  MoveL 1318 to (27.18, 67.36, -94.62) mm, rotated rx -11.83 ry -17.7 rz 126.62 deg; joints [8.101, -41.729, 125.318, 236.035, 70.646, -43.276, 143.741]
  MoveL 1319 to (26.72, 68.02, -94.62) mm, rotated rx -11.83 ry -17.7 rz 126.62 deg; joints [8.127, -41.741, 125.362, 236.053, 70.666, -43.25, 143.741]
  MoveL 1320 to (26.37, 68.63, -94.62) mm, rotated rx -11.83 ry -17.7 rz 126.62 deg; joints [8.149, -41.755, 125.404, 236.067, 70.684, -43.226, 143.741]
  MoveL 1321 to (26.15, 69.22, -94.62) mm, rotated rx -11.83 ry -17.7 rz 126.62 deg; joints [8.165, -41.771, 125.447, 236.075, 70.7, -43.204, 143.741]
  MoveL 1322 to (25.94, 69.86, -94.6) mm, rotated rx -11.83 ry -17.7 rz 126.62 deg; joints [8.181, -41.791, 125.494, 236.083, 70.717, -43.181, 143.741]
  MoveL 1323 to (25.74, 70.59, -94.56) mm, rotated rx -11.83 ry -17.7 rz 126.62 deg; joints [8.198, -41.815, 125.548, 236.092, 70.735, -43.156, 143.741]
  MoveL 1324 to (25.25, 72.63, -94.56) mm, rotated rx -11.83 ry -17.7 rz 126.62 deg; joints [8.24, -41.878, 125.7, 236.109, 70.789, -43.08, 143.741]
  MoveL 1325 to (25.13, 73.06, -94.54) mm, rotated rx -11.83 ry -17.7 rz 126.62 deg; joints [8.25, -41.892, 125.732, 236.114, 70.799, -43.066, 143.741]
  MoveL 1326 to (24.89, 74.08, -94.54) mm, rotated rx -11.83 ry -17.7 rz 126.62 deg; joints [8.271, -41.924, 125.808, 236.122, 70.826, -43.028, 143.741]
  MoveL 1327 to (24.77, 74.57, -94.54) mm, rotated rx -11.83 ry -17.7 rz 126.62 deg; joints [8.281, -41.939, 125.844, 236.127, 70.839, -43.01, 143.741]
  MoveL 1328 to (24.64, 75.04, -94.52) mm, rotated rx -11.83 ry -17.7 rz 126.62 deg; joints [8.292, -41.954, 125.879, 236.132, 70.85, -42.993, 143.741]
  MoveL 1329 to (24.51, 75.5, -94.49) mm, rotated rx -11.83 ry -17.7 rz 126.62 deg; joints [8.303, -41.97, 125.913, 236.138, 70.862, -42.978, 143.741]
  MoveL 1330 to (24.37, 75.91, -94.43) mm, rotated rx -11.83 ry -17.7 rz 126.62 deg; joints [8.314, -41.985, 125.942, 236.145, 70.871, -42.966, 143.741]
  MoveL 1331 to (24.24, 76.37, -94.39) mm, rotated rx -11.83 ry -17.7 rz 126.62 deg; joints [8.325, -42, 125.975, 236.151, 70.882, -42.951, 143.741]
  MoveL 1332 to (24.11, 76.85, -94.37) mm, rotated rx -11.83 ry -17.7 rz 126.62 deg; joints [8.336, -42.016, 126.011, 236.156, 70.893, -42.935, 143.741]
  MoveL 1333 to (23.99, 77.34, -94.37) mm, rotated rx -11.83 ry -17.7 rz 126.62 deg; joints [8.347, -42.031, 126.047, 236.161, 70.906, -42.917, 143.741]
  MoveL 1334 to (23.86, 77.81, -94.35) mm, rotated rx -11.83 ry -17.7 rz 126.62 deg; joints [8.357, -42.047, 126.082, 236.167, 70.918, -42.9, 143.741]
  MoveL 1335 to (23.72, 78.27, -94.31) mm, rotated rx -11.83 ry -17.7 rz 126.62 deg; joints [8.369, -42.062, 126.116, 236.173, 70.929, -42.885, 143.741]
  MoveL 1336 to (23.58, 78.68, -94.26) mm, rotated rx -11.83 ry -17.7 rz 126.62 deg; joints [8.38, -42.077, 126.145, 236.18, 70.938, -42.873, 143.741]
  MoveL 1337 to (23.43, 79.11, -94.2) mm, rotated rx -11.83 ry -17.7 rz 126.62 deg; joints [8.392, -42.092, 126.176, 236.188, 70.948, -42.86, 143.741]
  MoveL 1338 to (23.03, 80.5, -94.12) mm, rotated rx -11.83 ry -17.7 rz 126.62 deg; joints [8.425, -42.138, 126.277, 236.205, 70.982, -42.813, 143.741]
  MoveL 1339 to (22.85, 81.66, -94.25) mm, rotated rx -11.83 ry -17.7 rz 126.62 deg; joints [8.443, -42.168, 126.366, 236.208, 71.015, -42.763, 143.741]
  MoveL 1340 to (22.88, 82.6, -94.58) mm, rotated rx -11.83 ry -17.7 rz 126.62 deg; joints [8.447, -42.184, 126.441, 236.194, 71.049, -42.711, 143.741]
  MoveL 1341 to (22.98, 82.99, -94.83) mm, rotated rx -11.83 ry -17.7 rz 126.62 deg; joints [8.444, -42.187, 126.475, 236.182, 71.066, -42.683, 143.741]
  MoveL 1342 to (23.13, 83.33, -95.13) mm, rotated rx -11.83 ry -17.7 rz 126.62 deg; joints [8.436, -42.185, 126.505, 236.165, 71.083, -42.655, 143.741]
  MoveL 1343 to (23.59, 83.83, -95.89) mm, rotated rx -11.83 ry -17.7 rz 126.62 deg; joints [8.41, -42.172, 126.556, 236.121, 71.116, -42.597, 143.741]
  MoveL 1344 to (24.27, 84.12, -96.86) mm, rotated rx -11.83 ry -17.7 rz 126.62 deg; joints [8.37, -42.143, 126.594, 236.061, 71.15, -42.536, 143.741]
  MoveL 1345 to (26.28, 84.03, -99.42) mm, rotated rx -11.83 ry -17.7 rz 126.62 deg; joints [8.244, -42.041, 126.632, 235.894, 71.219, -42.407, 143.741]
  MoveL 1346 to (28.47, 83.17, -102.03) mm, rotated rx -11.83 ry -17.7 rz 126.62 deg; joints [8.102, -41.913, 126.613, 235.72, 71.269, -42.304, 143.741]
  MoveL 1347 to (29.36, 82.49, -103.06) mm, rotated rx -11.83 ry -17.7 rz 126.62 deg; joints [8.041, -41.851, 126.579, 235.65, 71.28, -42.276, 143.741]
  MoveL 1348 to (30.13, 81.66, -103.9) mm, rotated rx -11.83 ry -17.7 rz 126.62 deg; joints [7.987, -41.791, 126.529, 235.592, 71.282, -42.264, 143.741]
  MoveL 1349 to (30.76, 80.65, -104.55) mm, rotated rx -11.83 ry -17.7 rz 126.62 deg; joints [7.94, -41.732, 126.464, 235.546, 71.275, -42.267, 143.741]
  MoveL 1350 to (31.27, 79.49, -105.02) mm, rotated rx -11.83 ry -17.7 rz 126.62 deg; joints [7.899, -41.675, 126.383, 235.511, 71.258, -42.286, 143.741]
  MoveL 1351 to (31.64, 78.15, -105.3) mm, rotated rx -11.83 ry -17.7 rz 126.62 deg; joints [7.865, -41.62, 126.286, 235.489, 71.232, -42.32, 143.741]
  MoveL 1352 to (31.88, 76.66, -105.39) mm, rotated rx -11.83 ry -17.7 rz 126.62 deg; joints [7.838, -41.566, 126.173, 235.478, 71.196, -42.37, 143.741]
  MoveL 1353 to (32.24, 73.52, -105.39) mm, rotated rx -11.83 ry -17.7 rz 126.62 deg; joints [7.791, -41.46, 125.932, 235.468, 71.116, -42.484, 143.741]
  MoveL 1354 to (32.31, 72.97, -105.41) mm, rotated rx -11.83 ry -17.7 rz 126.62 deg; joints [7.782, -41.441, 125.89, 235.466, 71.103, -42.504, 143.741]
  MoveL 1355 to (32.41, 72.36, -105.44) mm, rotated rx -11.83 ry -17.7 rz 126.62 deg; joints [7.772, -41.418, 125.844, 235.462, 71.088, -42.524, 143.741]
  MoveL 1356 to (32.55, 71.61, -105.54) mm, rotated rx -11.83 ry -17.7 rz 126.62 deg; joints [7.757, -41.389, 125.788, 235.454, 71.072, -42.547, 143.741]
  MoveL 1357 to (32.65, 71, -105.58) mm, rotated rx -11.83 ry -17.7 rz 126.62 deg; joints [7.746, -41.367, 125.741, 235.45, 71.057, -42.567, 143.741]
  MoveL 1358 to (32.72, 70.46, -105.59) mm, rotated rx -11.83 ry -17.7 rz 126.62 deg; joints [7.737, -41.348, 125.7, 235.447, 71.044, -42.586, 143.741]
  MoveL 1359 to (32.78, 69.96, -105.6) mm, rotated rx -11.83 ry -17.7 rz 126.62 deg; joints [7.729, -41.331, 125.662, 235.445, 71.031, -42.604, 143.741]
  MoveL 1360 to (32.85, 69.5, -105.61) mm, rotated rx -11.83 ry -17.7 rz 126.62 deg; joints [7.722, -41.315, 125.627, 235.443, 71.02, -42.62, 143.741]
  MoveL 1361 to (33.08, 67.46, -105.62) mm, rotated rx -11.83 ry -17.7 rz 126.62 deg; joints [7.691, -41.245, 125.47, 235.437, 70.968, -42.694, 143.741]
  MoveL 1362 to (33.16, 66.95, -105.66) mm, rotated rx -11.83 ry -17.7 rz 126.62 deg; joints [7.682, -41.227, 125.432, 235.433, 70.956, -42.711, 143.741]
  MoveL 1363 to (33.26, 66.49, -105.71) mm, rotated rx -11.83 ry -17.7 rz 126.62 deg; joints [7.673, -41.209, 125.397, 235.429, 70.945, -42.725, 143.741]
  MoveL 1364 to (33.36, 66.04, -105.78) mm, rotated rx -11.83 ry -17.7 rz 126.62 deg; joints [7.663, -41.191, 125.363, 235.423, 70.936, -42.738, 143.741]
  MoveL 1365 to (33.49, 65.57, -105.84) mm, rotated rx -11.83 ry -17.7 rz 126.62 deg; joints [7.652, -41.174, 125.329, 235.416, 70.925, -42.753, 143.741]
  MoveL 1366 to (33.66, 65.05, -105.88) mm, rotated rx -11.83 ry -17.7 rz 126.62 deg; joints [7.639, -41.157, 125.29, 235.41, 70.912, -42.771, 143.741]
  MoveL 1367 to (33.95, 64.44, -105.88) mm, rotated rx -11.83 ry -17.7 rz 126.62 deg; joints [7.62, -41.142, 125.247, 235.399, 70.894, -42.794, 143.741]
  MoveL 1368 to (34.35, 63.78, -105.88) mm, rotated rx -11.83 ry -17.7 rz 126.62 deg; joints [7.596, -41.128, 125.201, 235.383, 70.874, -42.82, 143.741]
  MoveL 1369 to (34.26, 65.71, -107.44) mm, rotated rx -11.83 ry -17.7 rz 126.62 deg; joints [7.597, -41.106, 125.358, 235.333, 70.976, -42.664, 143.741]
  MoveL 1370 to (35.81, 63.93, -107.57) mm, rotated rx -11.83 ry -17.7 rz 126.62 deg; joints [7.51, -41.073, 125.243, 235.268, 70.922, -42.731, 143.741]
  MoveL 1371 to (37.27, 62.24, -107.68) mm, rotated rx -11.83 ry -17.7 rz 126.62 deg; joints [7.428, -41.043, 125.134, 235.208, 70.869, -42.795, 143.741]
  MoveL 1372 to (38.69, 60.61, -107.84) mm, rotated rx -11.83 ry -17.7 rz 126.62 deg; joints [7.348, -41.012, 125.029, 235.148, 70.821, -42.854, 143.741]
  MoveL 1373 to (40.09, 59, -107.95) mm, rotated rx -11.83 ry -17.7 rz 126.62 deg; joints [7.27, -40.982, 124.924, 235.09, 70.771, -42.915, 143.741]
  MoveL 1374 to (41.49, 57.38, -108.06) mm, rotated rx -11.83 ry -17.7 rz 126.62 deg; joints [7.193, -40.953, 124.818, 235.033, 70.72, -42.976, 143.741]
  MoveL 1375 to (42.89, 55.78, -108.28) mm, rotated rx -11.83 ry -17.7 rz 126.62 deg; joints [7.113, -40.918, 124.713, 234.972, 70.674, -43.031, 143.741]
  MoveL 1376 to (44.29, 54.16, -108.5) mm, rotated rx -11.83 ry -17.7 rz 126.62 deg; joints [7.034, -40.881, 124.608, 234.912, 70.627, -43.085, 143.741]
  MoveL 1377 to (45.68, 52.54, -108.62) mm, rotated rx -11.83 ry -17.7 rz 126.62 deg; joints [6.957, -40.851, 124.501, 234.856, 70.576, -43.146, 143.741]
  MoveL 1378 to (47.06, 50.91, -108.62) mm, rotated rx -11.83 ry -17.7 rz 126.62 deg; joints [6.882, -40.827, 124.393, 234.804, 70.521, -43.214, 143.741]
  MoveL 1379 to (48.44, 49.29, -108.73) mm, rotated rx -11.83 ry -17.7 rz 126.62 deg; joints [6.806, -40.796, 124.286, 234.748, 70.47, -43.275, 143.741]
  MoveL 1380 to (49.85, 47.65, -108.93) mm, rotated rx -11.83 ry -17.7 rz 126.62 deg; joints [6.727, -40.759, 124.177, 234.689, 70.421, -43.332, 143.741]
  MoveL 1381 to (51.15, 46.11, -109.11) mm, rotated rx -11.83 ry -17.7 rz 126.62 deg; joints [6.654, -40.725, 124.075, 234.635, 70.374, -43.386, 143.741]
  MoveL 1382 to (52.35, 44.7, -109.33) mm, rotated rx -11.83 ry -17.7 rz 126.62 deg; joints [6.587, -40.691, 123.981, 234.583, 70.334, -43.433, 143.741]
  MoveL 1383 to (53.63, 43.2, -109.42) mm, rotated rx -11.83 ry -17.7 rz 126.62 deg; joints [6.517, -40.663, 123.881, 234.533, 70.285, -43.49, 143.741]
  MoveL 1384 to (54.98, 41.6, -109.43) mm, rotated rx -11.83 ry -17.7 rz 126.62 deg; joints [6.444, -40.637, 123.774, 234.483, 70.231, -43.555, 143.741]
  MoveL 1385 to (56.72, 39.52, -109.53) mm, rotated rx -11.83 ry -17.7 rz 126.62 deg; joints [6.35, -40.599, 123.634, 234.417, 70.163, -43.636, 143.741]
  MoveL 1386 to (58.02, 37.96, -109.74) mm, rotated rx -11.83 ry -17.7 rz 126.62 deg; joints [6.277, -40.561, 123.529, 234.363, 70.116, -43.689, 143.741]
  MoveL 1387 to (59.42, 36.26, -109.94) mm, rotated rx -11.83 ry -17.7 rz 126.62 deg; joints [6.199, -40.521, 123.413, 234.306, 70.064, -43.748, 143.741]
  MoveL 1388 to (60.7, 34.69, -110.23) mm, rotated rx -11.83 ry -17.7 rz 126.62 deg; joints [6.127, -40.479, 123.307, 234.251, 70.02, -43.797, 143.741]
  MoveL 1389 to (61.97, 33.17, -110.36) mm, rotated rx -11.83 ry -17.7 rz 126.62 deg; joints [6.058, -40.446, 123.204, 234.201, 69.971, -43.853, 143.741]
  MoveL 1390 to (63.32, 31.57, -110.38) mm, rotated rx -11.83 ry -17.7 rz 126.62 deg; joints [5.986, -40.42, 123.095, 234.152, 69.916, -43.918, 143.741]
  MoveL 1391 to (64.43, 30.19, -110.6) mm, rotated rx -11.83 ry -17.7 rz 126.62 deg; joints [5.924, -40.382, 123, 234.106, 69.876, -43.963, 143.741]
  Set speed (1000.0 mm/s)
  MoveL 1392 to (88.04, 19.17, -110.6) mm, rotated rx -11.83 ry -17.7 rz 126.62 deg; joints [4.825, -40.56, 122.428, 233.209, 69.312, -44.514, 143.741]
  Set speed (1000.0 mm/s)
  MoveL 1393 to (85.28, 13.25, -121.79) mm, rotated rx -11.83 ry -17.7 rz 126.62 deg; joints [4.742, -39.632, 121.949, 232.99, 69.573, -44.122, 143.741]
  Set speed (100.0 mm/s)
  MoveL 1394 to (67, 21.77, -121.79) mm, rotated rx -11.83 ry -17.7 rz 126.62 deg; joints [5.589, -39.492, 122.393, 233.681, 70.009, -43.693, 143.741]
  MoveL 1395 to (65.84, 23.56, -121.79) mm, rotated rx -11.83 ry -17.7 rz 126.62 deg; joints [5.653, -39.53, 122.521, 233.72, 70.068, -43.62, 143.741]
  MoveL 1396 to (64.64, 25.44, -121.69) mm, rotated rx -11.83 ry -17.7 rz 126.62 deg; joints [5.721, -39.575, 122.656, 233.764, 70.128, -43.55, 143.741]
  MoveL 1397 to (63.4, 27.44, -121.4) mm, rotated rx -11.83 ry -17.7 rz 126.62 deg; joints [5.795, -39.635, 122.798, 233.814, 70.183, -43.484, 143.741]
  MoveL 1398 to (62.23, 29.36, -121.05) mm, rotated rx -11.83 ry -17.7 rz 126.62 deg; joints [5.866, -39.697, 122.935, 233.865, 70.234, -43.425, 143.741]
  MoveL 1399 to (61.12, 31.11, -120.86) mm, rotated rx -11.83 ry -17.7 rz 126.62 deg; joints [5.93, -39.745, 123.059, 233.909, 70.286, -43.364, 143.741]
  MoveL 1400 to (60.07, 32.75, -120.73) mm, rotated rx -11.83 ry -17.7 rz 126.62 deg; joints [5.991, -39.787, 123.175, 233.949, 70.335, -43.305, 143.741]
  MoveL 1401 to (58.95, 34.47, -120.68) mm, rotated rx -11.83 ry -17.7 rz 126.62 deg; joints [6.055, -39.825, 123.297, 233.99, 70.39, -43.238, 143.741]
  MoveL 1402 to (57.78, 36.26, -120.66) mm, rotated rx -11.83 ry -17.7 rz 126.62 deg; joints [6.12, -39.862, 123.423, 234.031, 70.448, -43.167, 143.741]
  MoveL 1403 to (56.63, 38.04, -120.54) mm, rotated rx -11.83 ry -17.7 rz 126.62 deg; joints [6.187, -39.905, 123.548, 234.075, 70.502, -43.101, 143.741]
  MoveL 1404 to (55.38, 39.96, -120.28) mm, rotated rx -11.83 ry -17.7 rz 126.62 deg; joints [6.261, -39.959, 123.682, 234.127, 70.556, -43.036, 143.741]
  MoveL 1405 to (54.07, 41.97, -120.09) mm, rotated rx -11.83 ry -17.7 rz 126.62 deg; joints [6.338, -40.01, 123.823, 234.18, 70.615, -42.965, 143.741]
  MoveL 1406 to (52.79, 43.92, -119.89) mm, rotated rx -11.83 ry -17.7 rz 126.62 deg; joints [6.413, -40.061, 123.959, 234.232, 70.672, -42.896, 143.741]
  MoveL 1407 to (51.62, 45.7, -119.78) mm, rotated rx -11.83 ry -17.7 rz 126.62 deg; joints [6.481, -40.103, 124.083, 234.278, 70.726, -42.83, 143.741]
  MoveL 1408 to (49.29, 49.23, -119.51) mm, rotated rx -11.83 ry -17.7 rz 126.62 deg; joints [6.618, -40.187, 124.328, 234.371, 70.83, -42.701, 143.741]
  MoveL 1409 to (48.1, 51.05, -119.44) mm, rotated rx -11.83 ry -17.7 rz 126.62 deg; joints [6.687, -40.227, 124.454, 234.417, 70.887, -42.631, 143.741]
  MoveL 1410 to (46.91, 52.82, -119.22) mm, rotated rx -11.83 ry -17.7 rz 126.62 deg; joints [6.758, -40.273, 124.575, 234.468, 70.936, -42.571, 143.741]
  MoveL 1411 to (45.73, 54.57, -119.06) mm, rotated rx -11.83 ry -17.7 rz 126.62 deg; joints [6.828, -40.316, 124.696, 234.517, 70.987, -42.508, 143.741]
  MoveL 1412 to (44.55, 56.32, -118.87) mm, rotated rx -11.83 ry -17.7 rz 126.62 deg; joints [6.898, -40.359, 124.816, 234.567, 71.036, -42.446, 143.741]
  MoveL 1413 to (43.34, 58.13, -118.78) mm, rotated rx -11.83 ry -17.7 rz 126.62 deg; joints [6.969, -40.399, 124.94, 234.615, 71.091, -42.377, 143.741]
  MoveL 1414 to (42.07, 60.01, -118.65) mm, rotated rx -11.83 ry -17.7 rz 126.62 deg; joints [7.044, -40.441, 125.068, 234.667, 71.147, -42.308, 143.741]
  MoveL 1415 to (41.03, 61.61, -118.59) mm, rotated rx -11.83 ry -17.7 rz 126.62 deg; joints [7.105, -40.476, 125.178, 234.708, 71.195, -42.246, 143.741]
  MoveL 1416 to (40.47, 61.24, -117.71) mm, rotated rx -11.83 ry -17.7 rz 126.62 deg; joints [7.138, -40.5, 125.138, 234.76, 71.16, -42.303, 143.741]
  MoveL 1417 to (40.45, 60.88, -117.3) mm, rotated rx -11.83 ry -17.7 rz 126.62 deg; joints [7.142, -40.511, 125.108, 234.775, 71.137, -42.339, 143.741]
  MoveL 1418 to (40.41, 60.83, -117.02) mm, rotated rx -11.83 ry -17.7 rz 126.62 deg; joints [7.147, -40.524, 125.102, 234.785, 71.126, -42.356, 143.741]
  MoveL 1419 to (40.36, 61.15, -116.9) mm, rotated rx -11.83 ry -17.7 rz 126.62 deg; joints [7.154, -40.542, 125.127, 234.79, 71.131, -42.35, 143.741]
  MoveL 1420 to (40.33, 61.6, -116.84) mm, rotated rx -11.83 ry -17.7 rz 126.62 deg; joints [7.16, -40.561, 125.162, 234.792, 71.141, -42.337, 143.741]
  MoveL 1421 to (40.31, 62.16, -116.81) mm, rotated rx -11.83 ry -17.7 rz 126.62 deg; joints [7.167, -40.583, 125.206, 234.793, 71.154, -42.318, 143.741]
  MoveL 1422 to (40.3, 62.86, -116.77) mm, rotated rx -11.83 ry -17.7 rz 126.62 deg; joints [7.175, -40.61, 125.26, 234.793, 71.17, -42.295, 143.741]
  MoveL 1423 to (40.29, 63.49, -116.74) mm, rotated rx -11.83 ry -17.7 rz 126.62 deg; joints [7.181, -40.634, 125.31, 234.793, 71.185, -42.273, 143.741]
  MoveL 1424 to (40.3, 64.02, -116.74) mm, rotated rx -11.83 ry -17.7 rz 126.62 deg; joints [7.186, -40.654, 125.352, 234.791, 71.199, -42.254, 143.741]
  MoveL 1425 to (40.29, 64.5, -116.73) mm, rotated rx -11.83 ry -17.7 rz 126.62 deg; joints [7.191, -40.672, 125.39, 234.791, 71.21, -42.237, 143.741]
  MoveL 1426 to (40.25, 65.54, -116.65) mm, rotated rx -11.83 ry -17.7 rz 126.62 deg; joints [7.204, -40.714, 125.471, 234.793, 71.234, -42.204, 143.741]
  MoveL 1427 to (40.22, 66.1, -116.6) mm, rotated rx -11.83 ry -17.7 rz 126.62 deg; joints [7.211, -40.736, 125.515, 234.794, 71.247, -42.186, 143.741]
  MoveL 1428 to (40.18, 66.61, -116.53) mm, rotated rx -11.83 ry -17.7 rz 126.62 deg; joints [7.218, -40.758, 125.554, 234.797, 71.258, -42.171, 143.741]
  MoveL 1429 to (40.14, 67.07, -116.46) mm, rotated rx -11.83 ry -17.7 rz 126.62 deg; joints [7.226, -40.778, 125.59, 234.8, 71.267, -42.158, 143.741]
  MoveL 1430 to (40.1, 67.54, -116.4) mm, rotated rx -11.83 ry -17.7 rz 126.62 deg; joints [7.232, -40.797, 125.625, 234.802, 71.277, -42.144, 143.741]
  MoveL 1431 to (40.09, 68.02, -116.37) mm, rotated rx -11.83 ry -17.7 rz 126.62 deg; joints [7.238, -40.816, 125.663, 234.803, 71.288, -42.129, 143.741]
  MoveL 1432 to (40.08, 68.54, -116.35) mm, rotated rx -11.83 ry -17.7 rz 126.62 deg; joints [7.244, -40.836, 125.704, 234.803, 71.301, -42.111, 143.741]
  MoveL 1433 to (40.12, 72.21, -116.35) mm, rotated rx -11.83 ry -17.7 rz 126.62 deg; joints [7.277, -40.971, 125.994, 234.793, 71.393, -41.979, 143.741]
  MoveL 1434 to (40.25, 73.83, -116.37) mm, rotated rx -11.83 ry -17.7 rz 126.62 deg; joints [7.286, -41.031, 126.123, 234.784, 71.433, -41.92, 143.741]
  MoveL 1435 to (40.39, 74.39, -116.4) mm, rotated rx -11.83 ry -17.7 rz 126.62 deg; joints [7.285, -41.054, 126.169, 234.776, 71.447, -41.899, 143.741]
  MoveL 1436 to (40.57, 74.79, -116.43) mm, rotated rx -11.83 ry -17.7 rz 126.62 deg; joints [7.281, -41.071, 126.204, 234.767, 71.456, -41.884, 143.741]
  MoveL 1437 to (40.78, 75.06, -116.47) mm, rotated rx -11.83 ry -17.7 rz 126.62 deg; joints [7.273, -41.084, 126.229, 234.756, 71.462, -41.874, 143.741]
  MoveL 1438 to (40.9, 75.14, -116.5) mm, rotated rx -11.83 ry -17.7 rz 126.62 deg; joints [7.268, -41.089, 126.237, 234.75, 71.464, -41.87, 143.741]
  MoveL 1439 to (41.03, 75.19, -116.52) mm, rotated rx -11.83 ry -17.7 rz 126.62 deg; joints [7.262, -41.093, 126.243, 234.744, 71.465, -41.868, 143.741]
  MoveL 1440 to (41.17, 75.22, -116.55) mm, rotated rx -11.83 ry -17.7 rz 126.62 deg; joints [7.256, -41.095, 126.247, 234.737, 71.466, -41.867, 143.741]
  MoveL 1441 to (41.31, 75.21, -116.58) mm, rotated rx -11.83 ry -17.7 rz 126.62 deg; joints [7.249, -41.097, 126.249, 234.73, 71.465, -41.866, 143.741]
  MoveL 1442 to (41.61, 75.13, -116.64) mm, rotated rx -11.83 ry -17.7 rz 126.62 deg; joints [7.234, -41.099, 126.248, 234.716, 71.462, -41.868, 143.741]
  MoveL 1443 to (42.28, 74.69, -116.77) mm, rotated rx -11.83 ry -17.7 rz 126.62 deg; joints [7.199, -41.093, 126.224, 234.685, 71.45, -41.882, 143.741]
  MoveL 1444 to (42.99, 73.98, -116.91) mm, rotated rx -11.83 ry -17.7 rz 126.62 deg; joints [7.158, -41.078, 126.18, 234.652, 71.43, -41.905, 143.741]
  MoveL 1445 to (44.42, 72.12, -117.18) mm, rotated rx -11.83 ry -17.7 rz 126.62 deg; joints [7.074, -41.033, 126.057, 234.587, 71.379, -41.967, 143.741]
  MoveL 1446 to (45.76, 70.11, -117.42) mm, rotated rx -11.83 ry -17.7 rz 126.62 deg; joints [6.992, -40.981, 125.921, 234.528, 71.324, -42.035, 143.741]
  MoveL 1447 to (75.42, 25.01, -122.5) mm, rotated rx -11.83 ry -17.7 rz 126.62 deg; joints [5.243, -39.788, 122.773, 233.304, 70.024, -43.595, 143.741]
  MoveL 1448 to (77.53, 21.81, -122.86) mm, rotated rx -11.83 ry -17.7 rz 126.62 deg; joints [5.123, -39.7, 122.543, 233.223, 69.927, -43.706, 143.741]
  MoveL 1449 to (79.44, 18.58, -123.28) mm, rotated rx -11.83 ry -17.7 rz 126.62 deg; joints [5.011, -39.603, 122.309, 233.149, 69.834, -43.814, 143.741]
  MoveL 1450 to (79.95, 17.18, -123.49) mm, rotated rx -11.83 ry -17.7 rz 126.62 deg; joints [4.975, -39.551, 122.203, 233.129, 69.798, -43.857, 143.741]
  MoveL 1451 to (79.98, 16.64, -123.58) mm, rotated rx -11.83 ry -17.7 rz 126.62 deg; joints [4.968, -39.526, 122.16, 233.127, 69.786, -43.872, 143.741]
  MoveL 1452 to (79.94, 16.41, -123.63) mm, rotated rx -11.83 ry -17.7 rz 126.62 deg; joints [4.968, -39.513, 122.141, 233.129, 69.783, -43.877, 143.741]
  MoveL 1453 to (79.84, 16.23, -123.67) mm, rotated rx -11.83 ry -17.7 rz 126.62 deg; joints [4.971, -39.502, 122.125, 233.132, 69.78, -43.881, 143.741]
  MoveL 1454 to (79.68, 16.09, -123.71) mm, rotated rx -11.83 ry -17.7 rz 126.62 deg; joints [4.976, -39.49, 122.112, 233.138, 69.78, -43.883, 143.741]
  MoveL 1455 to (79.47, 16, -123.74) mm, rotated rx -11.83 ry -17.7 rz 126.62 deg; joints [4.983, -39.479, 122.101, 233.146, 69.781, -43.883, 143.741]
  MoveL 1456 to (79.19, 15.95, -123.77) mm, rotated rx -11.83 ry -17.7 rz 126.62 deg; joints [4.994, -39.469, 122.094, 233.156, 69.784, -43.882, 143.741]
  MoveL 1457 to (78.85, 15.96, -123.8) mm, rotated rx -11.83 ry -17.7 rz 126.62 deg; joints [5.009, -39.459, 122.09, 233.169, 69.789, -43.878, 143.741]
  MoveL 1458 to (76.76, 16.59, -123.85) mm, rotated rx -11.83 ry -17.7 rz 126.62 deg; joints [5.103, -39.428, 122.114, 233.249, 69.831, -43.838, 143.741]
  MoveL 1459 to (74.83, 17.41, -123.85) mm, rotated rx -11.83 ry -17.7 rz 126.62 deg; joints [5.191, -39.41, 122.154, 233.322, 69.875, -43.796, 143.741]
  MoveL 1460 to (71.53, 19.31, -123.89) mm, rotated rx -11.83 ry -17.7 rz 126.62 deg; joints [5.346, -39.395, 122.263, 233.444, 69.964, -43.703, 143.741]
  MoveL 1461 to (68.92, 21.71, -124) mm, rotated rx -11.83 ry -17.7 rz 126.62 deg; joints [5.475, -39.413, 122.42, 233.534, 70.061, -43.593, 143.741]
  MoveL 1462 to (65.6, 26.76, -124.3) mm, rotated rx -11.83 ry -17.7 rz 126.62 deg; joints [5.654, -39.5, 122.782, 233.637, 70.241, -43.372, 143.741]
  MoveL 1463 to (64.74, 28.96, -124.43) mm, rotated rx -11.83 ry -17.7 rz 126.62 deg; joints [5.707, -39.553, 122.947, 233.658, 70.312, -43.279, 143.741]
  MoveL 1464 to (53.48, 61.86, -126.3) mm, rotated rx -11.83 ry -17.7 rz 126.62 deg; joints [6.45, -40.357, 125.41, 233.947, 71.352, -41.909, 143.741]
  MoveL 1465 to (52.5, 64.67, -126.46) mm, rotated rx -11.83 ry -17.7 rz 126.62 deg; joints [6.516, -40.423, 125.618, 233.975, 71.44, -41.791, 143.741]
  MoveL 1466 to (50.86, 68.02, -126.7) mm, rotated rx -11.83 ry -17.7 rz 126.62 deg; joints [6.615, -40.485, 125.858, 234.028, 71.551, -41.645, 143.741]
  MoveL 1467 to (49.92, 69.17, -126.84) mm, rotated rx -11.83 ry -17.7 rz 126.62 deg; joints [6.665, -40.493, 125.935, 234.06, 71.595, -41.589, 143.741]
  MoveL 1468 to (49.47, 69.48, -126.91) mm, rotated rx -11.83 ry -17.7 rz 126.62 deg; joints [6.687, -40.488, 125.952, 234.076, 71.609, -41.57, 143.741]
  MoveL 1469 to (49.25, 69.54, -126.94) mm, rotated rx -11.83 ry -17.7 rz 126.62 deg; joints [6.697, -40.482, 125.954, 234.084, 71.614, -41.565, 143.741]
  MoveL 1470 to (49.04, 69.55, -126.98) mm, rotated rx -11.83 ry -17.7 rz 126.62 deg; joints [6.706, -40.474, 125.951, 234.092, 71.618, -41.561, 143.741]
  MoveL 1471 to (48.84, 69.48, -127.01) mm, rotated rx -11.83 ry -17.7 rz 126.62 deg; joints [6.713, -40.465, 125.943, 234.099, 71.619, -41.56, 143.741]
  MoveL 1472 to (48.66, 69.34, -127.05) mm, rotated rx -11.83 ry -17.7 rz 126.62 deg; joints [6.72, -40.453, 125.929, 234.106, 71.619, -41.562, 143.741]
  MoveL 1473 to (48.48, 69.13, -127.08) mm, rotated rx -11.83 ry -17.7 rz 126.62 deg; joints [6.725, -40.438, 125.909, 234.113, 71.616, -41.567, 143.741]
  MoveL 1474 to (48.32, 68.82, -127.12) mm, rotated rx -11.83 ry -17.7 rz 126.62 deg; joints [6.729, -40.421, 125.883, 234.12, 71.611, -41.575, 143.741]
  MoveL 1475 to (47.84, 66.68, -127.24) mm, rotated rx -11.83 ry -17.7 rz 126.62 deg; joints [6.729, -40.324, 125.707, 234.141, 71.564, -41.642, 143.741]
  MoveL 1476 to (47.78, 66.17, -127.26) mm, rotated rx -11.83 ry -17.7 rz 126.62 deg; joints [6.727, -40.303, 125.665, 234.144, 71.552, -41.659, 143.741]
  MoveL 1477 to (47.76, 65.71, -127.31) mm, rotated rx -11.83 ry -17.7 rz 126.62 deg; joints [6.723, -40.283, 125.629, 234.145, 71.542, -41.673, 143.741]
  MoveL 1478 to (47.75, 65.27, -127.38) mm, rotated rx -11.83 ry -17.7 rz 126.62 deg; joints [6.718, -40.263, 125.594, 234.144, 71.534, -41.686, 143.741]
  MoveL 1479 to (47.73, 64.83, -127.44) mm, rotated rx -11.83 ry -17.7 rz 126.62 deg; joints [6.714, -40.243, 125.559, 234.144, 71.524, -41.699, 143.741]
  MoveL 1480 to (47.69, 64.36, -127.47) mm, rotated rx -11.83 ry -17.7 rz 126.62 deg; joints [6.711, -40.223, 125.522, 234.146, 71.514, -41.713, 143.741]
  MoveL 1481 to (47.05, 59.72, -127.48) mm, rotated rx -11.83 ry -17.7 rz 126.62 deg; joints [6.698, -40.039, 125.145, 234.184, 71.4, -41.877, 143.741]
  MoveL 1482 to (47.01, 59.28, -127.5) mm, rotated rx -11.83 ry -17.7 rz 126.62 deg; joints [6.695, -40.021, 125.109, 234.186, 71.39, -41.892, 143.741]
  MoveL 1483 to (46.95, 58.81, -127.51) mm, rotated rx -11.83 ry -17.7 rz 126.62 deg; joints [6.694, -40.002, 125.071, 234.19, 71.378, -41.908, 143.741]
  MoveL 1484 to (46.81, 57.79, -127.52) mm, rotated rx -11.83 ry -17.7 rz 126.62 deg; joints [6.691, -39.961, 124.987, 234.198, 71.353, -41.945, 143.741]
  MoveL 1485 to (46.74, 57.22, -127.52) mm, rotated rx -11.83 ry -17.7 rz 126.62 deg; joints [6.688, -39.938, 124.941, 234.203, 71.339, -41.965, 143.741]
  MoveL 1486 to (46.69, 56.62, -127.54) mm, rotated rx -11.83 ry -17.7 rz 126.62 deg; joints [6.685, -39.914, 124.893, 234.206, 71.325, -41.985, 143.741]
  MoveL 1487 to (46.67, 55.95, -127.57) mm, rotated rx -11.83 ry -17.7 rz 126.62 deg; joints [6.679, -39.888, 124.84, 234.207, 71.309, -42.008, 143.741]
  MoveL 1488 to (46.73, 55.29, -127.59) mm, rotated rx -11.83 ry -17.7 rz 126.62 deg; joints [6.671, -39.864, 124.789, 234.206, 71.292, -42.031, 143.741]
  MoveL 1489 to (46.84, 54.65, -127.61) mm, rotated rx -11.83 ry -17.7 rz 126.62 deg; joints [6.66, -39.843, 124.739, 234.203, 71.275, -42.055, 143.741]
  MoveL 1490 to (46.91, 55.96, -128.59) mm, rotated rx -11.83 ry -17.7 rz 126.62 deg; joints [6.655, -39.834, 124.846, 234.166, 71.342, -41.955, 143.741]
  MoveL 1491 to (47.76, 54.93, -129.02) mm, rotated rx -11.83 ry -17.7 rz 126.62 deg; joints [6.602, -39.794, 124.779, 234.12, 71.322, -41.976, 143.741]
  MoveL 1492 to (48.61, 53.7, -129.33) mm, rotated rx -11.83 ry -17.7 rz 126.62 deg; joints [6.549, -39.753, 124.695, 234.078, 71.293, -42.01, 143.741]
  MoveL 1493 to (49.47, 52.24, -129.57) mm, rotated rx -11.83 ry -17.7 rz 126.62 deg; joints [6.495, -39.71, 124.593, 234.04, 71.255, -42.057, 143.741]
  MoveL 1494 to (50.45, 50.34, -129.79) mm, rotated rx -11.83 ry -17.7 rz 126.62 deg; joints [6.432, -39.654, 124.457, 233.998, 71.204, -42.122, 143.741]
  MoveL 1495 to (51.4, 48.43, -129.9) mm, rotated rx -11.83 ry -17.7 rz 126.62 deg; joints [6.373, -39.603, 124.32, 233.961, 71.149, -42.192, 143.741]
  MoveL 1496 to (52.35, 46.52, -130.01) mm, rotated rx -11.83 ry -17.7 rz 126.62 deg; joints [6.313, -39.552, 124.182, 233.925, 71.093, -42.263, 143.741]
  MoveL 1497 to (53.31, 44.62, -130.24) mm, rotated rx -11.83 ry -17.7 rz 126.62 deg; joints [6.251, -39.495, 124.045, 233.884, 71.041, -42.327, 143.741]
  MoveL 1498 to (54.26, 42.7, -130.36) mm, rotated rx -11.83 ry -17.7 rz 126.62 deg; joints [6.192, -39.443, 123.907, 233.848, 70.986, -42.397, 143.741]
  MoveL 1499 to (55.21, 40.79, -130.59) mm, rotated rx -11.83 ry -17.7 rz 126.62 deg; joints [6.131, -39.385, 123.769, 233.808, 70.934, -42.461, 143.741]
  MoveL 1500 to (56.15, 38.88, -130.71) mm, rotated rx -11.83 ry -17.7 rz 126.62 deg; joints [6.072, -39.333, 123.63, 233.773, 70.878, -42.532, 143.741]
  MoveL 1501 to (57.09, 36.96, -130.82) mm, rotated rx -11.83 ry -17.7 rz 126.62 deg; joints [6.014, -39.28, 123.491, 233.738, 70.822, -42.602, 143.741]
  MoveL 1502 to (58.02, 35.04, -131.06) mm, rotated rx -11.83 ry -17.7 rz 126.62 deg; joints [5.954, -39.221, 123.352, 233.699, 70.77, -42.667, 143.741]
  MoveL 1503 to (58.91, 33.2, -131.17) mm, rotated rx -11.83 ry -17.7 rz 126.62 deg; joints [5.899, -39.17, 123.217, 233.667, 70.716, -42.735, 143.741]
  MoveL 1504 to (59.76, 31.41, -131.37) mm, rotated rx -11.83 ry -17.7 rz 126.62 deg; joints [5.844, -39.114, 123.086, 233.633, 70.667, -42.795, 143.741]
  MoveL 1505 to (60.81, 29.28, -131.53) mm, rotated rx -11.83 ry -17.7 rz 126.62 deg; joints [5.78, -39.054, 122.931, 233.594, 70.605, -42.872, 143.741]
  MoveL 1506 to (61.97, 26.82, -131.62) mm, rotated rx -11.83 ry -17.7 rz 126.62 deg; joints [5.708, -38.988, 122.749, 233.554, 70.53, -42.966, 143.741]
  MoveL 1507 to (62.87, 24.95, -131.69) mm, rotated rx -11.83 ry -17.7 rz 126.62 deg; joints [5.653, -38.938, 122.612, 233.523, 70.473, -43.037, 143.741]
  MoveL 1508 to (63.71, 23.22, -131.81) mm, rotated rx -11.83 ry -17.7 rz 126.62 deg; joints [5.602, -38.889, 122.485, 233.493, 70.422, -43.099, 143.741]
  MoveL 1509 to (64.57, 21.43, -131.92) mm, rotated rx -11.83 ry -17.7 rz 126.62 deg; joints [5.549, -38.838, 122.353, 233.463, 70.369, -43.165, 143.741]
  MoveL 1510 to (65.41, 19.67, -132.03) mm, rotated rx -11.83 ry -17.7 rz 126.62 deg; joints [5.498, -38.788, 122.223, 233.433, 70.317, -43.23, 143.741]
  MoveL 1511 to (66.3, 17.81, -132.1) mm, rotated rx -11.83 ry -17.7 rz 126.62 deg; joints [5.444, -38.738, 122.085, 233.404, 70.26, -43.3, 143.741]
  MoveL 1512 to (67.25, 15.8, -132.2) mm, rotated rx -11.83 ry -17.7 rz 126.62 deg; joints [5.386, -38.682, 121.937, 233.372, 70.199, -43.375, 143.741]
  MoveL 1513 to (68.26, 13.61, -132.46) mm, rotated rx -11.83 ry -17.7 rz 126.62 deg; joints [5.323, -38.611, 121.774, 233.334, 70.138, -43.449, 143.741]
  MoveL 1514 to (69.64, 11.85, -133.44) mm, rotated rx -11.83 ry -17.7 rz 126.62 deg; joints [5.236, -38.525, 121.652, 233.256, 70.109, -43.472, 143.741]
  MoveL 1515 to (68.66, 12.44, -133.93) mm, rotated rx -11.83 ry -17.7 rz 126.62 deg; joints [5.276, -38.494, 121.687, 233.277, 70.152, -43.42, 143.741]
  MoveL 1516 to (68.15, 12.74, -134.24) mm, rotated rx -11.83 ry -17.7 rz 126.62 deg; joints [5.296, -38.475, 121.705, 233.287, 70.176, -43.389, 143.741]
  MoveL 1517 to (68.06, 12.79, -134.39) mm, rotated rx -11.83 ry -17.7 rz 126.62 deg; joints [5.298, -38.466, 121.707, 233.285, 70.183, -43.379, 143.741]
  MoveL 1518 to (68.36, 12.61, -134.43) mm, rotated rx -11.83 ry -17.7 rz 126.62 deg; joints [5.283, -38.464, 121.697, 233.273, 70.176, -43.386, 143.741]
  MoveL 1519 to (68.76, 12.37, -134.44) mm, rotated rx -11.83 ry -17.7 rz 126.62 deg; joints [5.264, -38.465, 121.683, 233.258, 70.166, -43.397, 143.741]
  MoveL 1520 to (69.16, 12.11, -134.48) mm, rotated rx -11.83 ry -17.7 rz 126.62 deg; joints [5.244, -38.463, 121.668, 233.242, 70.156, -43.407, 143.741]
  MoveL 1521 to (69.53, 11.85, -134.54) mm, rotated rx -11.83 ry -17.7 rz 126.62 deg; joints [5.226, -38.46, 121.652, 233.226, 70.147, -43.416, 143.741]
  MoveL 1522 to (69.92, 11.6, -134.58) mm, rotated rx -11.83 ry -17.7 rz 126.62 deg; joints [5.207, -38.457, 121.637, 233.211, 70.137, -43.426, 143.741]
  MoveL 1523 to (70.33, 11.34, -134.6) mm, rotated rx -11.83 ry -17.7 rz 126.62 deg; joints [5.187, -38.457, 121.622, 233.195, 70.126, -43.437, 143.741]
  MoveL 1524 to (72.6, 10.02, -134.6) mm, rotated rx -11.83 ry -17.7 rz 126.62 deg; joints [5.08, -38.465, 121.546, 233.11, 70.066, -43.5, 143.741]
  MoveL 1525 to (72.98, 9.78, -134.62) mm, rotated rx -11.83 ry -17.7 rz 126.62 deg; joints [5.061, -38.465, 121.532, 233.095, 70.056, -43.511, 143.741]
  MoveL 1526 to (73.31, 9.56, -134.65) mm, rotated rx -11.83 ry -17.7 rz 126.62 deg; joints [5.046, -38.463, 121.519, 233.082, 70.047, -43.519, 143.741]
  MoveL 1527 to (73.7, 9.32, -134.67) mm, rotated rx -11.83 ry -17.7 rz 126.62 deg; joints [5.027, -38.463, 121.504, 233.067, 70.037, -43.529, 143.741]
  MoveL 1528 to (74.2, 9, -134.69) mm, rotated rx -11.83 ry -17.7 rz 126.62 deg; joints [5.003, -38.462, 121.486, 233.048, 70.024, -43.543, 143.741]
  MoveL 1529 to (74.81, 8.61, -134.75) mm, rotated rx -11.83 ry -17.7 rz 126.62 deg; joints [4.973, -38.46, 121.462, 233.024, 70.008, -43.559, 143.741]
  MoveL 1530 to (75.33, 8.28, -134.78) mm, rotated rx -11.83 ry -17.7 rz 126.62 deg; joints [4.948, -38.459, 121.442, 233.004, 69.994, -43.573, 143.741]
  MoveL 1531 to (75.79, 8.01, -134.78) mm, rotated rx -11.83 ry -17.7 rz 126.62 deg; joints [4.926, -38.46, 121.426, 232.987, 69.982, -43.586, 143.741]
  MoveL 1532 to (77.15, 7.22, -134.78) mm, rotated rx -11.83 ry -17.7 rz 126.62 deg; joints [4.863, -38.465, 121.38, 232.937, 69.945, -43.624, 143.741]
  MoveL 1533 to (79.5, 5.5, -135.12) mm, rotated rx -11.83 ry -17.7 rz 126.62 deg; joints [4.745, -38.44, 121.273, 232.841, 69.883, -43.685, 143.741]
  MoveL 1534 to (80.39, 4.56, -135.55) mm, rotated rx -11.83 ry -17.7 rz 126.62 deg; joints [4.695, -38.403, 121.208, 232.797, 69.862, -43.704, 143.741]
  MoveL 1535 to (81.09, 3.56, -136.15) mm, rotated rx -11.83 ry -17.7 rz 126.62 deg; joints [4.649, -38.349, 121.137, 232.757, 69.847, -43.715, 143.741]
  MoveL 1536 to (81.89, 1.38, -137.86) mm, rotated rx -11.83 ry -17.7 rz 126.62 deg; joints [4.576, -38.191, 120.972, 232.683, 69.836, -43.714, 143.741]
  MoveL 1537 to (81.93, -1.03, -140.26) mm, rotated rx -11.83 ry -17.7 rz 126.62 deg; joints [4.523, -37.966, 120.779, 232.621, 69.85, -43.684, 143.741]
  MoveL 1538 to (81.31, -2.99, -142.65) mm, rotated rx -11.83 ry -17.7 rz 126.62 deg; joints [4.502, -37.743, 120.613, 232.583, 69.882, -43.633, 143.741]
  MoveL 1539 to (80.79, -3.55, -143.59) mm, rotated rx -11.83 ry -17.7 rz 126.62 deg; joints [4.507, -37.656, 120.561, 232.577, 69.904, -43.604, 143.741]
  MoveL 1540 to (80.15, -3.84, -144.36) mm, rotated rx -11.83 ry -17.7 rz 126.62 deg; joints [4.522, -37.586, 120.53, 232.581, 69.929, -43.572, 143.741]
  MoveL 1541 to (79.77, -3.88, -144.68) mm, rotated rx -11.83 ry -17.7 rz 126.62 deg; joints [4.533, -37.557, 120.522, 232.586, 69.943, -43.556, 143.741]
  MoveL 1542 to (79.36, -3.85, -144.96) mm, rotated rx -11.83 ry -17.7 rz 126.62 deg; joints [4.547, -37.532, 120.519, 232.594, 69.958, -43.538, 143.741]
  MoveL 1543 to (78.44, -3.57, -145.39) mm, rotated rx -11.83 ry -17.7 rz 126.62 deg; joints [4.581, -37.495, 120.529, 232.616, 69.99, -43.501, 143.741]
  MoveL 1544 to (77.39, -3.02, -145.65) mm, rotated rx -11.83 ry -17.7 rz 126.62 deg; joints [4.626, -37.475, 120.56, 232.647, 70.025, -43.461, 143.741]
  MoveL 1545 to (76.2, -2.19, -145.73) mm, rotated rx -11.83 ry -17.7 rz 126.62 deg; joints [4.682, -37.471, 120.612, 232.687, 70.064, -43.418, 143.741]
  MoveL 1546 to (75.78, -1.88, -145.73) mm, rotated rx -11.83 ry -17.7 rz 126.62 deg; joints [4.702, -37.472, 120.633, 232.702, 70.077, -43.404, 143.741]
  MoveL 1547 to (75.46, -1.58, -145.68) mm, rotated rx -11.83 ry -17.7 rz 126.62 deg; joints [4.718, -37.478, 120.653, 232.715, 70.087, -43.393, 143.741]
  MoveL 1548 to (75.14, -1.28, -145.62) mm, rotated rx -11.83 ry -17.7 rz 126.62 deg; joints [4.735, -37.485, 120.672, 232.727, 70.097, -43.383, 143.741]
  MoveL 1549 to (74.78, -0.97, -145.58) mm, rotated rx -11.83 ry -17.7 rz 126.62 deg; joints [4.753, -37.489, 120.693, 232.741, 70.108, -43.371, 143.741]
  MoveL 1550 to (74.4, -0.66, -145.56) mm, rotated rx -11.83 ry -17.7 rz 126.62 deg; joints [4.771, -37.492, 120.713, 232.755, 70.121, -43.358, 143.741]
  MoveL 1551 to (73.98, -0.33, -145.56) mm, rotated rx -11.83 ry -17.7 rz 126.62 deg; joints [4.792, -37.495, 120.734, 232.771, 70.134, -43.343, 143.741]
  MoveL 1552 to (73.56, -0.01, -145.56) mm, rotated rx -11.83 ry -17.7 rz 126.62 deg; joints [4.812, -37.496, 120.755, 232.785, 70.147, -43.329, 143.741]
  MoveL 1553 to (73.15, 0.29, -145.57) mm, rotated rx -11.83 ry -17.7 rz 126.62 deg; joints [4.831, -37.496, 120.773, 232.8, 70.161, -43.314, 143.741]
  MoveL 1554 to (72.75, 0.58, -145.58) mm, rotated rx -11.83 ry -17.7 rz 126.62 deg; joints [4.85, -37.496, 120.792, 232.814, 70.174, -43.3, 143.741]
  MoveL 1555 to (72.39, 0.87, -145.56) mm, rotated rx -11.83 ry -17.7 rz 126.62 deg; joints [4.868, -37.499, 120.811, 232.827, 70.185, -43.288, 143.741]
  MoveL 1556 to (72.04, 1.18, -145.52) mm, rotated rx -11.83 ry -17.7 rz 126.62 deg; joints [4.885, -37.504, 120.83, 232.841, 70.196, -43.276, 143.741]
  MoveL 1557 to (71.63, 1.53, -145.47) mm, rotated rx -11.83 ry -17.7 rz 126.62 deg; joints [4.906, -37.509, 120.854, 232.857, 70.208, -43.263, 143.741]
  MoveL 1558 to (71.1, 2, -145.42) mm, rotated rx -11.83 ry -17.7 rz 126.62 deg; joints [4.933, -37.516, 120.884, 232.877, 70.225, -43.245, 143.741]
  MoveL 1559 to (70.6, 2.41, -145.4) mm, rotated rx -11.83 ry -17.7 rz 126.62 deg; joints [4.957, -37.52, 120.911, 232.896, 70.241, -43.228, 143.741]
  MoveL 1560 to (68.53, 4, -145.4) mm, rotated rx -11.83 ry -17.7 rz 126.62 deg; joints [5.058, -37.527, 121.012, 232.971, 70.307, -43.155, 143.741]
  MoveL 1561 to (68.04, 4.4, -145.36) mm, rotated rx -11.83 ry -17.7 rz 126.62 deg; joints [5.082, -37.531, 121.037, 232.989, 70.322, -43.139, 143.741]
  MoveL 1562 to (67.62, 4.76, -145.3) mm, rotated rx -11.83 ry -17.7 rz 126.62 deg; joints [5.103, -37.537, 121.061, 233.007, 70.334, -43.126, 143.741]
  MoveL 1563 to (67.46, 4.9, -145.15) mm, rotated rx -11.83 ry -17.7 rz 126.62 deg; joints [5.113, -37.547, 121.07, 233.017, 70.335, -43.127, 143.741]
  MoveL 1564 to (67.55, 4.82, -144.89) mm, rotated rx -11.83 ry -17.7 rz 126.62 deg; joints [5.112, -37.561, 121.064, 233.021, 70.323, -43.144, 143.741]
  MoveL 1565 to (67.89, 4.52, -144.48) mm, rotated rx -11.83 ry -17.7 rz 126.62 deg; joints [5.101, -37.582, 121.044, 233.022, 70.297, -43.177, 143.741]
  MoveL 1566 to (68.24, 5.49, -143.68) mm, rotated rx -11.83 ry -17.7 rz 126.62 deg; joints [5.105, -37.671, 121.127, 233.028, 70.293, -43.183, 143.741]
  MoveL 1567 to (67.66, 7.38, -143.46) mm, rotated rx -11.83 ry -17.7 rz 126.62 deg; joints [5.147, -37.739, 121.273, 233.048, 70.344, -43.12, 143.741]
  MoveL 1568 to (67.05, 9.29, -143.3) mm, rotated rx -11.83 ry -17.7 rz 126.62 deg; joints [5.189, -37.803, 121.42, 233.068, 70.398, -43.053, 143.741]
  MoveL 1569 to (66.42, 11.25, -143.15) mm, rotated rx -11.83 ry -17.7 rz 126.62 deg; joints [5.233, -37.867, 121.57, 233.088, 70.453, -42.983, 143.741]
  MoveL 1570 to (65.86, 13.04, -142.86) mm, rotated rx -11.83 ry -17.7 rz 126.62 deg; joints [5.275, -37.935, 121.707, 233.111, 70.498, -42.928, 143.741]
  MoveL 1571 to (65.21, 15.05, -142.67) mm, rotated rx -11.83 ry -17.7 rz 126.62 deg; joints [5.321, -38.003, 121.86, 233.134, 70.554, -42.858, 143.741]
  MoveL 1572 to (64.53, 17.16, -142.49) mm, rotated rx -11.83 ry -17.7 rz 126.62 deg; joints [5.369, -38.073, 122.021, 233.157, 70.612, -42.785, 143.741]
  MoveL 1573 to (63.83, 19.29, -142.4) mm, rotated rx -11.83 ry -17.7 rz 126.62 deg; joints [5.417, -38.138, 122.183, 233.178, 70.674, -42.705, 143.741]
  MoveL 1574 to (62.97, 21.88, -142.31) mm, rotated rx -11.83 ry -17.7 rz 126.62 deg; joints [5.476, -38.216, 122.38, 233.204, 70.75, -42.608, 143.741]
  MoveL 1575 to (62.35, 23.74, -142.21) mm, rotated rx -11.83 ry -17.7 rz 126.62 deg; joints [5.519, -38.273, 122.52, 233.225, 70.804, -42.54, 143.741]
  MoveL 1576 to (61.77, 25.47, -141.99) mm, rotated rx -11.83 ry -17.7 rz 126.62 deg; joints [5.56, -38.334, 122.651, 233.248, 70.849, -42.483, 143.741]
  MoveL 1577 to (61.13, 27.38, -141.8) mm, rotated rx -11.83 ry -17.7 rz 126.62 deg; joints [5.606, -38.397, 122.796, 233.272, 70.901, -42.417, 143.741]
  MoveL 1578 to (60.44, 29.4, -141.68) mm, rotated rx -11.83 ry -17.7 rz 126.62 deg; joints [5.654, -38.46, 122.948, 233.295, 70.959, -42.344, 143.741]
  MoveL 1579 to (59.76, 31.4, -141.5) mm, rotated rx -11.83 ry -17.7 rz 126.62 deg; joints [5.702, -38.525, 123.099, 233.32, 71.014, -42.274, 143.741]
  MoveL 1580 to (59.08, 33.4, -141.38) mm, rotated rx -11.83 ry -17.7 rz 126.62 deg; joints [5.749, -38.586, 123.249, 233.344, 71.07, -42.202, 143.741]
  MoveL 1581 to (58.37, 35.46, -141.2) mm, rotated rx -11.83 ry -17.7 rz 126.62 deg; joints [5.8, -38.652, 123.404, 233.371, 71.127, -42.13, 143.741]
  MoveL 1582 to (57.67, 37.48, -141.08) mm, rotated rx -11.83 ry -17.7 rz 126.62 deg; joints [5.848, -38.714, 123.555, 233.395, 71.184, -42.056, 143.741]
  MoveL 1583 to (56.96, 39.49, -140.85) mm, rotated rx -11.83 ry -17.7 rz 126.62 deg; joints [5.899, -38.781, 123.705, 233.424, 71.237, -41.989, 143.741]
  MoveL 1584 to (56.26, 41.51, -140.74) mm, rotated rx -11.83 ry -17.7 rz 126.62 deg; joints [5.948, -38.842, 123.856, 233.449, 71.294, -41.915, 143.741]
  MoveL 1585 to (55.56, 43.53, -140.62) mm, rotated rx -11.83 ry -17.7 rz 126.62 deg; joints [5.997, -38.902, 124.006, 233.475, 71.351, -41.842, 143.741]
  MoveL 1586 to (54.83, 45.54, -140.4) mm, rotated rx -11.83 ry -17.7 rz 126.62 deg; joints [6.049, -38.968, 124.155, 233.505, 71.404, -41.774, 143.741]
  MoveL 1587 to (54.12, 47.34, -140.19) mm, rotated rx -11.83 ry -17.7 rz 126.62 deg; joints [6.098, -39.026, 124.288, 233.534, 71.452, -41.713, 143.741]
  MoveL 1588 to (53.42, 48.96, -139.9) mm, rotated rx -11.83 ry -17.7 rz 126.62 deg; joints [6.147, -39.083, 124.406, 233.567, 71.491, -41.663, 143.741]
  MoveL 1589 to (52.7, 50.42, -139.5) mm, rotated rx -11.83 ry -17.7 rz 126.62 deg; joints [6.197, -39.14, 124.511, 233.605, 71.523, -41.625, 143.741]
  MoveL 1590 to (52.66, 48.93, -138.57) mm, rotated rx -11.83 ry -17.7 rz 126.62 deg; joints [6.199, -39.141, 124.391, 233.64, 71.451, -41.728, 143.741]
  MoveL 1591 to (52.59, 49.51, -138.56) mm, rotated rx -11.83 ry -17.7 rz 126.62 deg; joints [6.208, -39.16, 124.436, 233.641, 71.467, -41.707, 143.741]
  MoveL 1592 to (52.56, 50.04, -138.54) mm, rotated rx -11.83 ry -17.7 rz 126.62 deg; joints [6.214, -39.18, 124.478, 233.641, 71.481, -41.688, 143.741]
  MoveL 1593 to (52.58, 50.51, -138.48) mm, rotated rx -11.83 ry -17.7 rz 126.62 deg; joints [6.218, -39.2, 124.515, 233.641, 71.491, -41.674, 143.741]
  MoveL 1594 to (52.62, 50.96, -138.41) mm, rotated rx -11.83 ry -17.7 rz 126.62 deg; joints [6.221, -39.221, 124.551, 233.64, 71.5, -41.661, 143.741]
  MoveL 1595 to (52.7, 51.41, -138.36) mm, rotated rx -11.83 ry -17.7 rz 126.62 deg; joints [6.222, -39.243, 124.589, 233.637, 71.51, -41.648, 143.741]
  MoveL 1596 to (52.8, 51.89, -138.33) mm, rotated rx -11.83 ry -17.7 rz 126.62 deg; joints [6.222, -39.264, 124.628, 233.632, 71.52, -41.632, 143.741]
  MoveL 1597 to (52.93, 52.4, -138.31) mm, rotated rx -11.83 ry -17.7 rz 126.62 deg; joints [6.221, -39.287, 124.671, 233.626, 71.532, -41.615, 143.741]
  MoveL 1598 to (53.06, 52.91, -138.31) mm, rotated rx -11.83 ry -17.7 rz 126.62 deg; joints [6.219, -39.308, 124.713, 233.618, 71.544, -41.598, 143.741]
  MoveL 1599 to (53.18, 53.36, -138.3) mm, rotated rx -11.83 ry -17.7 rz 126.62 deg; joints [6.219, -39.328, 124.751, 233.613, 71.555, -41.582, 143.741]
  MoveL 1600 to (53.26, 53.78, -138.28) mm, rotated rx -11.83 ry -17.7 rz 126.62 deg; joints [6.219, -39.347, 124.785, 233.609, 71.564, -41.569, 143.741]
  MoveL 1601 to (53.38, 54.24, -138.26) mm, rotated rx -11.83 ry -17.7 rz 126.62 deg; joints [6.218, -39.367, 124.824, 233.603, 71.575, -41.553, 143.741]
  MoveL 1602 to (53.52, 54.75, -138.26) mm, rotated rx -11.83 ry -17.7 rz 126.62 deg; joints [6.216, -39.389, 124.866, 233.596, 71.587, -41.536, 143.741]
  MoveL 1603 to (53.67, 55.34, -138.24) mm, rotated rx -11.83 ry -17.7 rz 126.62 deg; joints [6.215, -39.415, 124.916, 233.588, 71.601, -41.516, 143.741]
  MoveL 1604 to (53.83, 56.02, -138.2) mm, rotated rx -11.83 ry -17.7 rz 126.62 deg; joints [6.214, -39.446, 124.972, 233.581, 71.616, -41.495, 143.741]
  MoveL 1605 to (53.98, 56.61, -138.18) mm, rotated rx -11.83 ry -17.7 rz 126.62 deg; joints [6.213, -39.472, 125.021, 233.573, 71.63, -41.475, 143.741]
  MoveL 1606 to (54.13, 57.23, -138.15) mm, rotated rx -11.83 ry -17.7 rz 126.62 deg; joints [6.212, -39.499, 125.072, 233.566, 71.644, -41.455, 143.741]
  MoveL 1607 to (54.28, 57.93, -138.12) mm, rotated rx -11.83 ry -17.7 rz 126.62 deg; joints [6.212, -39.53, 125.13, 233.559, 71.66, -41.432, 143.741]
  MoveL 1608 to (54.43, 58.5, -138.1) mm, rotated rx -11.83 ry -17.7 rz 126.62 deg; joints [6.211, -39.555, 125.177, 233.551, 71.673, -41.413, 143.741]
  MoveL 1609 to (54.57, 59.02, -138.1) mm, rotated rx -11.83 ry -17.7 rz 126.62 deg; joints [6.209, -39.578, 125.221, 233.544, 71.686, -41.395, 143.741]
  MoveL 1610 to (54.98, 60.54, -138.1) mm, rotated rx -11.83 ry -17.7 rz 126.62 deg; joints [6.204, -39.642, 125.348, 233.522, 71.722, -41.342, 143.741]
  MoveL 1611 to (55.43, 61.92, -138.18) mm, rotated rx -11.83 ry -17.7 rz 126.62 deg; joints [6.195, -39.698, 125.464, 233.497, 71.757, -41.29, 143.741]
  MoveL 1612 to (55.94, 63, -138.44) mm, rotated rx -11.83 ry -17.7 rz 126.62 deg; joints [6.178, -39.734, 125.557, 233.465, 71.79, -41.242, 143.741]
  MoveL 1613 to (56.5, 63.77, -138.86) mm, rotated rx -11.83 ry -17.7 rz 126.62 deg; joints [6.153, -39.75, 125.627, 233.426, 71.821, -41.195, 143.741]
  MoveL 1614 to (56.81, 64.04, -139.13) mm, rotated rx -11.83 ry -17.7 rz 126.62 deg; joints [6.138, -39.752, 125.653, 233.404, 71.835, -41.173, 143.741]
  MoveL 1615 to (57.13, 64.23, -139.45) mm, rotated rx -11.83 ry -17.7 rz 126.62 deg; joints [6.121, -39.748, 125.674, 233.38, 71.848, -41.152, 143.741]
  MoveL 1616 to (57.82, 64.4, -140.21) mm, rotated rx -11.83 ry -17.7 rz 126.62 deg; joints [6.081, -39.726, 125.698, 233.328, 71.873, -41.111, 143.741]
  MoveL 1617 to (58.56, 64.26, -141.14) mm, rotated rx -11.83 ry -17.7 rz 126.62 deg; joints [6.033, -39.684, 125.698, 233.268, 71.896, -41.074, 143.741]
  MoveL 1618 to (60.24, 63.06, -143.5) mm, rotated rx -11.83 ry -17.7 rz 126.62 deg; joints [5.915, -39.543, 125.631, 233.129, 71.933, -41.007, 143.741]
  MoveL 1619 to (61.66, 61.12, -145.86) mm, rotated rx -11.83 ry -17.7 rz 126.62 deg; joints [5.801, -39.37, 125.499, 233.004, 71.953, -40.966, 143.741]
  MoveL 1620 to (62.32, 58.89, -147.55) mm, rotated rx -11.83 ry -17.7 rz 126.62 deg; joints [5.729, -39.207, 125.333, 232.931, 71.947, -40.966, 143.741]
  MoveL 1621 to (62.37, 57.67, -148.14) mm, rotated rx -11.83 ry -17.7 rz 126.62 deg; joints [5.708, -39.13, 125.238, 232.915, 71.934, -40.981, 143.741]
  MoveL 1622 to (62.23, 56.38, -148.56) mm, rotated rx -11.83 ry -17.7 rz 126.62 deg; joints [5.697, -39.056, 125.133, 232.912, 71.915, -41.006, 143.741]
  MoveL 1623 to (61.38, 53.59, -148.9) mm, rotated rx -11.83 ry -17.7 rz 126.62 deg; joints [5.707, -38.916, 124.899, 232.947, 71.859, -41.085, 143.741]
  MoveL 1624 to (59.77, 49.73, -148.9) mm, rotated rx -11.83 ry -17.7 rz 126.62 deg; joints [5.746, -38.739, 124.568, 233.027, 71.769, -41.217, 143.741]
  MoveL 1625 to (59.57, 49.21, -148.92) mm, rotated rx -11.83 ry -17.7 rz 126.62 deg; joints [5.75, -38.715, 124.524, 233.036, 71.757, -41.233, 143.741]
  MoveL 1626 to (59.4, 48.72, -148.96) mm, rotated rx -11.83 ry -17.7 rz 126.62 deg; joints [5.753, -38.69, 124.482, 233.044, 71.747, -41.248, 143.741]
  MoveL 1627 to (59.23, 48.21, -149.02) mm, rotated rx -11.83 ry -17.7 rz 126.62 deg; joints [5.756, -38.664, 124.439, 233.05, 71.737, -41.263, 143.741]
  MoveL 1628 to (59.09, 47.71, -149.1) mm, rotated rx -11.83 ry -17.7 rz 126.62 deg; joints [5.757, -38.638, 124.398, 233.056, 71.727, -41.276, 143.741]
  MoveL 1629 to (58.94, 47.23, -149.18) mm, rotated rx -11.83 ry -17.7 rz 126.62 deg; joints [5.758, -38.613, 124.357, 233.061, 71.718, -41.289, 143.741]
  MoveL 1630 to (58.78, 46.77, -149.22) mm, rotated rx -11.83 ry -17.7 rz 126.62 deg; joints [5.761, -38.59, 124.318, 233.068, 71.709, -41.303, 143.741]
  MoveL 1631 to (58.61, 46.32, -149.23) mm, rotated rx -11.83 ry -17.7 rz 126.62 deg; joints [5.764, -38.569, 124.28, 233.076, 71.699, -41.317, 143.741]
  MoveL 1632 to (58.41, 45.84, -149.23) mm, rotated rx -11.83 ry -17.7 rz 126.62 deg; joints [5.769, -38.547, 124.238, 233.086, 71.687, -41.334, 143.741]
  MoveL 1633 to (58.19, 45.25, -149.27) mm, rotated rx -11.83 ry -17.7 rz 126.62 deg; joints [5.774, -38.519, 124.188, 233.097, 71.674, -41.352, 143.741]
  MoveL 1634 to (57.96, 44.61, -149.33) mm, rotated rx -11.83 ry -17.7 rz 126.62 deg; joints [5.777, -38.486, 124.133, 233.106, 71.661, -41.371, 143.741]
  MoveL 1635 to (57.77, 44.04, -149.35) mm, rotated rx -11.83 ry -17.7 rz 126.62 deg; joints [5.781, -38.461, 124.085, 233.116, 71.648, -41.39, 143.741]
  MoveL 1636 to (57.62, 43.51, -149.36) mm, rotated rx -11.83 ry -17.7 rz 126.62 deg; joints [5.783, -38.437, 124.04, 233.123, 71.635, -41.409, 143.741]
  MoveL 1637 to (57.53, 42.96, -149.36) mm, rotated rx -11.83 ry -17.7 rz 126.62 deg; joints [5.782, -38.416, 123.995, 233.129, 71.621, -41.428, 143.741]
  MoveL 1638 to (57.55, 42.39, -149.36) mm, rotated rx -11.83 ry -17.7 rz 126.62 deg; joints [5.776, -38.396, 123.95, 233.13, 71.605, -41.45, 143.741]
  MoveL 1639 to (57.65, 41.78, -149.36) mm, rotated rx -11.83 ry -17.7 rz 126.62 deg; joints [5.767, -38.377, 123.903, 233.128, 71.588, -41.473, 143.741]
  MoveL 1640 to (57.77, 43.35, -150.32) mm, rotated rx -11.83 ry -17.7 rz 126.62 deg; joints [5.761, -38.378, 124.03, 233.089, 71.663, -41.367, 143.741]
  MoveL 1641 to (58.23, 42.2, -150.74) mm, rotated rx -11.83 ry -17.7 rz 126.62 deg; joints [5.725, -38.325, 123.945, 233.061, 71.642, -41.391, 143.741]
  MoveL 1642 to (58.66, 40.85, -151.07) mm, rotated rx -11.83 ry -17.7 rz 126.62 deg; joints [5.691, -38.269, 123.843, 233.038, 71.612, -41.428, 143.741]
  MoveL 1643 to (59.07, 39.29, -151.32) mm, rotated rx -11.83 ry -17.7 rz 126.62 deg; joints [5.657, -38.21, 123.725, 233.019, 71.575, -41.476, 143.741]
  MoveL 1644 to (59.51, 37.2, -151.43) mm, rotated rx -11.83 ry -17.7 rz 126.62 deg; joints [5.619, -38.142, 123.565, 233.006, 71.517, -41.552, 143.741]
  MoveL 1645 to (59.97, 35.12, -151.66) mm, rotated rx -11.83 ry -17.7 rz 126.62 deg; joints [5.579, -38.066, 123.405, 232.988, 71.463, -41.621, 143.741]
  MoveL 1646 to (60.4, 33.04, -151.77) mm, rotated rx -11.83 ry -17.7 rz 126.62 deg; joints [5.542, -37.997, 123.244, 232.975, 71.406, -41.697, 143.741]
  MoveL 1647 to (60.83, 30.95, -151.89) mm, rotated rx -11.83 ry -17.7 rz 126.62 deg; joints [5.505, -37.927, 123.082, 232.962, 71.348, -41.772, 143.741]
  MoveL 1648 to (61.27, 28.86, -152.13) mm, rotated rx -11.83 ry -17.7 rz 126.62 deg; joints [5.466, -37.851, 122.921, 232.945, 71.294, -41.841, 143.741]
  MoveL 1649 to (61.7, 26.77, -152.25) mm, rotated rx -11.83 ry -17.7 rz 126.62 deg; joints [5.429, -37.781, 122.759, 232.933, 71.236, -41.916, 143.741]
  MoveL 1650 to (62.12, 24.68, -152.36) mm, rotated rx -11.83 ry -17.7 rz 126.62 deg; joints [5.393, -37.71, 122.597, 232.921, 71.179, -41.992, 143.741]
  MoveL 1651 to (62.61, 22.27, -152.52) mm, rotated rx -11.83 ry -17.7 rz 126.62 deg; joints [5.35, -37.628, 122.41, 232.906, 71.112, -42.077, 143.741]
  MoveL 1652 to (63.02, 20.21, -152.72) mm, rotated rx -11.83 ry -17.7 rz 126.62 deg; joints [5.314, -37.553, 122.25, 232.893, 71.058, -42.148, 143.741]
  MoveL 1653 to (63.47, 17.94, -152.92) mm, rotated rx -11.83 ry -17.7 rz 126.62 deg; joints [5.274, -37.472, 122.073, 232.878, 70.997, -42.226, 143.741]
  MoveL 1654 to (63.9, 15.72, -153.17) mm, rotated rx -11.83 ry -17.7 rz 126.62 deg; joints [5.235, -37.389, 121.9, 232.864, 70.94, -42.3, 143.741]
  MoveL 1655 to (64.31, 13.63, -153.29) mm, rotated rx -11.83 ry -17.7 rz 126.62 deg; joints [5.2, -37.317, 121.736, 232.853, 70.882, -42.375, 143.741]
  MoveL 1656 to (64.73, 11.54, -153.29) mm, rotated rx -11.83 ry -17.7 rz 126.62 deg; joints [5.166, -37.253, 121.572, 232.846, 70.819, -42.456, 143.741]
  MoveL 1657 to (65.13, 9.47, -153.37) mm, rotated rx -11.83 ry -17.7 rz 126.62 deg; joints [5.132, -37.184, 121.411, 232.838, 70.76, -42.533, 143.741]
  MoveL 1658 to (65.5, 7.45, -153.58) mm, rotated rx -11.83 ry -17.7 rz 126.62 deg; joints [5.098, -37.108, 121.251, 232.826, 70.707, -42.601, 143.741]
  MoveL 1659 to (65.89, 5.18, -153.93) mm, rotated rx -11.83 ry -17.7 rz 126.62 deg; joints [5.059, -37.016, 121.072, 232.811, 70.651, -42.672, 143.741]
  MoveL 1660 to (66.2, 3.4, -154.15) mm, rotated rx -11.83 ry -17.7 rz 126.62 deg; joints [5.03, -36.947, 120.932, 232.801, 70.606, -42.731, 143.741]
  MoveL 1661 to (66.6, 0.98, -154.44) mm, rotated rx -11.83 ry -17.7 rz 126.62 deg; joints [4.99, -36.853, 120.74, 232.789, 70.544, -42.81, 143.741]
  MoveL 1662 to (67, -1.2, -154.55) mm, rotated rx -11.83 ry -17.7 rz 126.62 deg; joints [4.956, -36.778, 120.568, 232.781, 70.482, -42.89, 143.741]
  MoveL 1663 to (67.41, -3.28, -154.56) mm, rotated rx -11.83 ry -17.7 rz 126.62 deg; joints [4.923, -36.712, 120.404, 232.775, 70.42, -42.97, 143.741]
  MoveL 1664 to (67.06, -4.11, -155.35) mm, rotated rx -11.83 ry -17.7 rz 126.62 deg; joints [4.921, -36.628, 120.331, 232.77, 70.426, -42.961, 143.741]
  MoveL 1665 to (66.82, -3.74, -155.74) mm, rotated rx -11.83 ry -17.7 rz 126.62 deg; joints [4.928, -36.613, 120.358, 232.766, 70.452, -42.927, 143.741]
  MoveL 1666 to (66.74, -3.62, -155.99) mm, rotated rx -11.83 ry -17.7 rz 126.62 deg; joints [4.929, -36.602, 120.366, 232.761, 70.464, -42.91, 143.741]
  MoveL 1667 to (66.84, -3.73, -156.11) mm, rotated rx -11.83 ry -17.7 rz 126.62 deg; joints [4.922, -36.594, 120.359, 232.754, 70.464, -42.908, 143.741]
  MoveL 1668 to (67.11, -4.01, -156.13) mm, rotated rx -11.83 ry -17.7 rz 126.62 deg; joints [4.908, -36.589, 120.339, 232.744, 70.454, -42.92, 143.741]
  MoveL 1669 to (67.44, -4.35, -156.14) mm, rotated rx -11.83 ry -17.7 rz 126.62 deg; joints [4.892, -36.584, 120.317, 232.732, 70.441, -42.934, 143.741]
  MoveL 1670 to (68.55, -5.46, -156.14) mm, rotated rx -11.83 ry -17.7 rz 126.62 deg; joints [4.837, -36.572, 120.241, 232.694, 70.399, -42.983, 143.741]
  MoveL 1671 to (68.93, -5.86, -156.16) mm, rotated rx -11.83 ry -17.7 rz 126.62 deg; joints [4.817, -36.565, 120.214, 232.68, 70.384, -42.999, 143.741]
  MoveL 1672 to (69.3, -6.27, -156.21) mm, rotated rx -11.83 ry -17.7 rz 126.62 deg; joints [4.798, -36.557, 120.185, 232.666, 70.37, -43.015, 143.741]
  MoveL 1673 to (69.66, -6.72, -156.29) mm, rotated rx -11.83 ry -17.7 rz 126.62 deg; joints [4.778, -36.545, 120.154, 232.652, 70.357, -43.03, 143.741]
  MoveL 1674 to (70.03, -7.13, -156.35) mm, rotated rx -11.83 ry -17.7 rz 126.62 deg; joints [4.759, -36.536, 120.125, 232.638, 70.343, -43.045, 143.741]
  MoveL 1675 to (70.39, -7.52, -156.37) mm, rotated rx -11.83 ry -17.7 rz 126.62 deg; joints [4.741, -36.529, 120.098, 232.624, 70.329, -43.061, 143.741]
  MoveL 1676 to (70.73, -7.88, -156.39) mm, rotated rx -11.83 ry -17.7 rz 126.62 deg; joints [4.723, -36.524, 120.074, 232.612, 70.316, -43.076, 143.741]
  MoveL 1677 to (71.03, -8.23, -156.44) mm, rotated rx -11.83 ry -17.7 rz 126.62 deg; joints [4.708, -36.516, 120.05, 232.601, 70.305, -43.088, 143.741]
  MoveL 1678 to (71.32, -8.56, -156.47) mm, rotated rx -11.83 ry -17.7 rz 126.62 deg; joints [4.692, -36.509, 120.027, 232.59, 70.294, -43.101, 143.741]
  MoveL 1679 to (71.67, -8.92, -156.49) mm, rotated rx -11.83 ry -17.7 rz 126.62 deg; joints [4.675, -36.504, 120.002, 232.578, 70.28, -43.116, 143.741]
  MoveL 1680 to (72.07, -9.34, -156.51) mm, rotated rx -11.83 ry -17.7 rz 126.62 deg; joints [4.655, -36.497, 119.973, 232.563, 70.265, -43.134, 143.741]
  MoveL 1681 to (72.54, -9.87, -156.56) mm, rotated rx -11.83 ry -17.7 rz 126.62 deg; joints [4.63, -36.486, 119.936, 232.546, 70.247, -43.154, 143.741]
  MoveL 1682 to (72.95, -10.31, -156.59) mm, rotated rx -11.83 ry -17.7 rz 126.62 deg; joints [4.609, -36.479, 119.905, 232.531, 70.231, -43.172, 143.741]
  MoveL 1683 to (74.44, -11.8, -156.59) mm, rotated rx -11.83 ry -17.7 rz 126.62 deg; joints [4.536, -36.461, 119.804, 232.481, 70.173, -43.237, 143.741]
  MoveL 1684 to (76.28, -14.05, -156.92) mm, rotated rx -11.83 ry -17.7 rz 126.62 deg; joints [4.438, -36.405, 119.644, 232.411, 70.1, -43.318, 143.741]
  MoveL 1685 to (76.91, -15.18, -157.33) mm, rotated rx -11.83 ry -17.7 rz 126.62 deg; joints [4.398, -36.356, 119.559, 232.38, 70.075, -43.345, 143.741]
  MoveL 1686 to (77.33, -16.32, -157.91) mm, rotated rx -11.83 ry -17.7 rz 126.62 deg; joints [4.364, -36.292, 119.47, 232.353, 70.057, -43.363, 143.741]
  MoveL 1687 to (77.58, -18.61, -159.56) mm, rotated rx -11.83 ry -17.7 rz 126.62 deg; joints [4.315, -36.122, 119.284, 232.307, 70.042, -43.372, 143.741]
  MoveL 1688 to (77.03, -20.93, -161.87) mm, rotated rx -11.83 ry -17.7 rz 126.62 deg; joints [4.291, -35.894, 119.085, 232.274, 70.057, -43.346, 143.741]
  MoveL 1689 to (75.95, -22.64, -164.17) mm, rotated rx -11.83 ry -17.7 rz 126.62 deg; joints [4.292, -35.675, 118.927, 232.258, 70.094, -43.296, 143.741]
  MoveL 1690 to (75.32, -23.05, -165.08) mm, rotated rx -11.83 ry -17.7 rz 126.62 deg; joints [4.303, -35.594, 118.884, 232.258, 70.119, -43.264, 143.741]
  MoveL 1691 to (74.63, -23.15, -165.82) mm, rotated rx -11.83 ry -17.7 rz 126.62 deg; joints [4.321, -35.532, 118.865, 232.264, 70.147, -43.229, 143.741]
  MoveL 1692 to (74.26, -23.09, -166.13) mm, rotated rx -11.83 ry -17.7 rz 126.62 deg; joints [4.333, -35.508, 118.865, 232.269, 70.163, -43.21, 143.741]
  MoveL 1693 to (73.88, -22.95, -166.4) mm, rotated rx -11.83 ry -17.7 rz 126.62 deg; joints [4.346, -35.488, 118.87, 232.276, 70.179, -43.19, 143.741]
  MoveL 1694 to (73.06, -22.45, -166.81) mm, rotated rx -11.83 ry -17.7 rz 126.62 deg; joints [4.378, -35.464, 118.9, 232.293, 70.216, -43.146, 143.741]
  MoveL 1695 to (72.18, -21.65, -167.06) mm, rotated rx -11.83 ry -17.7 rz 126.62 deg; joints [4.417, -35.457, 118.954, 232.315, 70.256, -43.098, 143.741]
  MoveL 1696 to (71.24, -20.54, -167.14) mm, rotated rx -11.83 ry -17.7 rz 126.62 deg; joints [4.463, -35.47, 119.032, 232.343, 70.3, -43.046, 143.741]
  MoveL 1697 to (69, -17.64, -167.14) mm, rotated rx -11.83 ry -17.7 rz 126.62 deg; joints [4.577, -35.519, 119.24, 232.415, 70.407, -42.922, 143.741]
  MoveL 1698 to (68.73, -17.27, -167.13) mm, rotated rx -11.83 ry -17.7 rz 126.62 deg; joints [4.592, -35.527, 119.267, 232.424, 70.42, -42.907, 143.741]
  MoveL 1699 to (68.49, -16.93, -167.1) mm, rotated rx -11.83 ry -17.7 rz 126.62 deg; joints [4.604, -35.535, 119.291, 232.433, 70.431, -42.894, 143.741]
  MoveL 1700 to (68.21, -16.55, -167.08) mm, rotated rx -11.83 ry -17.7 rz 126.62 deg; joints [4.619, -35.542, 119.319, 232.442, 70.444, -42.878, 143.741]
  MoveL 1701 to (65.97, -13.65, -167.08) mm, rotated rx -11.83 ry -17.7 rz 126.62 deg; joints [4.734, -35.591, 119.525, 232.515, 70.55, -42.753, 143.741]
  MoveL 1702 to (65.66, -13.21, -167.06) mm, rotated rx -11.83 ry -17.7 rz 126.62 deg; joints [4.751, -35.601, 119.557, 232.525, 70.565, -42.735, 143.741]
  MoveL 1703 to (65.37, -12.75, -167.02) mm, rotated rx -11.83 ry -17.7 rz 126.62 deg; joints [4.767, -35.612, 119.591, 232.535, 70.58, -42.717, 143.741]
  MoveL 1704 to (65.15, -12.31, -166.98) mm, rotated rx -11.83 ry -17.7 rz 126.62 deg; joints [4.78, -35.625, 119.624, 232.543, 70.594, -42.702, 143.741]
  MoveL 1705 to (65.01, -11.95, -166.92) mm, rotated rx -11.83 ry -17.7 rz 126.62 deg; joints [4.789, -35.638, 119.651, 232.549, 70.603, -42.69, 143.741]
  MoveL 1706 to (64.98, -11.76, -166.75) mm, rotated rx -11.83 ry -17.7 rz 126.62 deg; joints [4.794, -35.653, 119.667, 232.554, 70.603, -42.691, 143.741]
  MoveL 1707 to (65.01, -11.73, -166.42) mm, rotated rx -11.83 ry -17.7 rz 126.62 deg; joints [4.798, -35.673, 119.67, 232.562, 70.593, -42.705, 143.741]
  MoveL 1708 to (65.09, -11.87, -165.91) mm, rotated rx -11.83 ry -17.7 rz 126.62 deg; joints [4.801, -35.7, 119.66, 232.575, 70.572, -42.735, 143.741]
  MoveL 1709 to (65.6, -11.22, -164.45) mm, rotated rx -11.83 ry -17.7 rz 126.62 deg; joints [4.804, -35.819, 119.723, 232.594, 70.538, -42.783, 143.741]
  MoveL 1710 to (65.32, -6.96, -164.45) mm, rotated rx -11.83 ry -17.7 rz 126.62 deg; joints [4.847, -35.964, 120.067, 232.582, 70.662, -42.618, 143.741]
  MoveL 1711 to (65.19, -4.92, -164.4) mm, rotated rx -11.83 ry -17.7 rz 126.62 deg; joints [4.868, -36.037, 120.232, 232.578, 70.72, -42.542, 143.741]
  MoveL 1712 to (65.06, -2.95, -164.31) mm, rotated rx -11.83 ry -17.7 rz 126.62 deg; joints [4.889, -36.109, 120.392, 232.575, 70.775, -42.47, 143.741]
  MoveL 1713 to (64.93, -0.94, -164.23) mm, rotated rx -11.83 ry -17.7 rz 126.62 deg; joints [4.91, -36.183, 120.554, 232.572, 70.831, -42.396, 143.741]
  MoveL 1714 to (64.81, 1.03, -164.13) mm, rotated rx -11.83 ry -17.7 rz 126.62 deg; joints [4.931, -36.255, 120.713, 232.57, 70.885, -42.325, 143.741]
  MoveL 1715 to (64.69, 3.12, -164.09) mm, rotated rx -11.83 ry -17.7 rz 126.62 deg; joints [4.952, -36.329, 120.882, 232.565, 70.944, -42.247, 143.741]
  MoveL 1716 to (64.65, 5.32, -164.06) mm, rotated rx -11.83 ry -17.7 rz 126.62 deg; joints [4.971, -36.408, 121.06, 232.557, 71.006, -42.164, 143.741]
  MoveL 1717 to (64.4, 7.81, -163.89) mm, rotated rx -11.83 ry -17.7 rz 126.62 deg; joints [5.003, -36.499, 121.259, 232.56, 71.074, -42.076, 143.741]
  MoveL 1718 to (64.25, 10.04, -163.64) mm, rotated rx -11.83 ry -17.7 rz 126.62 deg; joints [5.029, -36.589, 121.439, 232.562, 71.13, -42.002, 143.741]
  MoveL 1719 to (64.1, 12.23, -163.51) mm, rotated rx -11.83 ry -17.7 rz 126.62 deg; joints [5.054, -36.671, 121.615, 232.561, 71.189, -41.924, 143.741]
  MoveL 1720 to (63.96, 14.36, -163.27) mm, rotated rx -11.83 ry -17.7 rz 126.62 deg; joints [5.08, -36.756, 121.785, 232.565, 71.243, -41.854, 143.741]
  MoveL 1721 to (63.81, 16.49, -163.15) mm, rotated rx -11.83 ry -17.7 rz 126.62 deg; joints [5.104, -36.834, 121.955, 232.564, 71.3, -41.779, 143.741]
  MoveL 1722 to (63.66, 18.62, -163.03) mm, rotated rx -11.83 ry -17.7 rz 126.62 deg; joints [5.128, -36.912, 122.125, 232.564, 71.358, -41.703, 143.741]
  MoveL 1723 to (63.49, 20.75, -162.79) mm, rotated rx -11.83 ry -17.7 rz 126.62 deg; joints [5.155, -36.997, 122.295, 232.569, 71.412, -41.633, 143.741]
  MoveL 1724 to (63.34, 22.87, -162.67) mm, rotated rx -11.83 ry -17.7 rz 126.62 deg; joints [5.18, -37.074, 122.465, 232.569, 71.469, -41.557, 143.741]
  MoveL 1725 to (63.18, 25, -162.55) mm, rotated rx -11.83 ry -17.7 rz 126.62 deg; joints [5.205, -37.151, 122.634, 232.57, 71.527, -41.481, 143.741]
  MoveL 1726 to (63.02, 27.13, -162.43) mm, rotated rx -11.83 ry -17.7 rz 126.62 deg; joints [5.23, -37.228, 122.803, 232.571, 71.584, -41.406, 143.741]
  MoveL 1727 to (62.83, 29.26, -162.2) mm, rotated rx -11.83 ry -17.7 rz 126.62 deg; joints [5.258, -37.311, 122.971, 232.577, 71.638, -41.335, 143.741]
  MoveL 1728 to (62.66, 31.38, -162.09) mm, rotated rx -11.83 ry -17.7 rz 126.62 deg; joints [5.283, -37.388, 123.14, 232.578, 71.695, -41.259, 143.741]
  MoveL 1729 to (62.48, 33.16, -161.84) mm, rotated rx -11.83 ry -17.7 rz 126.62 deg; joints [5.308, -37.46, 123.28, 232.586, 71.738, -41.203, 143.741]
  MoveL 1730 to (62.29, 34.8, -161.52) mm, rotated rx -11.83 ry -17.7 rz 126.62 deg; joints [5.334, -37.531, 123.409, 232.597, 71.775, -41.156, 143.741]
  MoveL 1731 to (62.09, 36.36, -161.1) mm, rotated rx -11.83 ry -17.7 rz 126.62 deg; joints [5.361, -37.605, 123.532, 232.612, 71.806, -41.117, 143.741]
  MoveL 1732 to (61.49, 34.73, -160.14) mm, rotated rx -11.83 ry -17.7 rz 126.62 deg; joints [5.389, -37.589, 123.393, 232.672, 71.732, -41.222, 143.741]
  MoveL 1733 to (61.49, 35.36, -160.02) mm, rotated rx -11.83 ry -17.7 rz 126.62 deg; joints [5.396, -37.619, 123.444, 232.673, 71.746, -41.204, 143.741]
  MoveL 1734 to (61.55, 35.94, -159.93) mm, rotated rx -11.83 ry -17.7 rz 126.62 deg; joints [5.398, -37.646, 123.491, 232.671, 71.758, -41.187, 143.741]
  MoveL 1735 to (61.72, 36.46, -159.9) mm, rotated rx -11.83 ry -17.7 rz 126.62 deg; joints [5.396, -37.67, 123.535, 232.663, 71.77, -41.171, 143.741]
  MoveL 1736 to (61.93, 36.95, -159.88) mm, rotated rx -11.83 ry -17.7 rz 126.62 deg; joints [5.391, -37.694, 123.577, 232.653, 71.781, -41.155, 143.741]
  MoveL 1737 to (63.75, 40.15, -159.87) mm, rotated rx -11.83 ry -17.7 rz 126.62 deg; joints [5.336, -37.852, 123.86, 232.565, 71.854, -41.048, 143.741]
  MoveL 1738 to (63.97, 40.56, -159.86) mm, rotated rx -11.83 ry -17.7 rz 126.62 deg; joints [5.33, -37.873, 123.896, 232.555, 71.863, -41.035, 143.741]
  MoveL 1739 to (64.16, 40.93, -159.83) mm, rotated rx -11.83 ry -17.7 rz 126.62 deg; joints [5.325, -37.892, 123.928, 232.546, 71.87, -41.024, 143.741]
  MoveL 1740 to (64.4, 41.35, -159.82) mm, rotated rx -11.83 ry -17.7 rz 126.62 deg; joints [5.318, -37.913, 123.965, 232.535, 71.88, -41.01, 143.741]
  MoveL 1741 to (64.66, 41.81, -159.82) mm, rotated rx -11.83 ry -17.7 rz 126.62 deg; joints [5.31, -37.936, 124.006, 232.523, 71.89, -40.995, 143.741]
  MoveL 1742 to (65.45, 43.17, -159.82) mm, rotated rx -11.83 ry -17.7 rz 126.62 deg; joints [5.286, -38.003, 124.126, 232.485, 71.921, -40.95, 143.741]
  MoveL 1743 to (65.75, 43.71, -159.8) mm, rotated rx -11.83 ry -17.7 rz 126.62 deg; joints [5.278, -38.031, 124.174, 232.471, 71.933, -40.933, 143.741]
  MoveL 1744 to (66.08, 44.35, -159.76) mm, rotated rx -11.83 ry -17.7 rz 126.62 deg; joints [5.269, -38.064, 124.229, 232.456, 71.946, -40.914, 143.741]
  MoveL 1745 to (66.39, 44.91, -159.74) mm, rotated rx -11.83 ry -17.7 rz 126.62 deg; joints [5.26, -38.093, 124.279, 232.442, 71.958, -40.896, 143.741]
  MoveL 1746 to (66.91, 45.82, -159.74) mm, rotated rx -11.83 ry -17.7 rz 126.62 deg; joints [5.244, -38.138, 124.359, 232.416, 71.979, -40.866, 143.741]
  MoveL 1747 to (67.69, 47.04, -159.83) mm, rotated rx -11.83 ry -17.7 rz 126.62 deg; joints [5.218, -38.195, 124.468, 232.377, 72.008, -40.822, 143.741]
  MoveL 1748 to (68.46, 47.95, -160.08) mm, rotated rx -11.83 ry -17.7 rz 126.62 deg; joints [5.187, -38.231, 124.551, 232.334, 72.036, -40.782, 143.741]
  MoveL 1749 to (69.2, 48.54, -160.5) mm, rotated rx -11.83 ry -17.7 rz 126.62 deg; joints [5.153, -38.245, 124.609, 232.288, 72.061, -40.744, 143.741]
  MoveL 1750 to (69.57, 48.73, -160.77) mm, rotated rx -11.83 ry -17.7 rz 126.62 deg; joints [5.134, -38.245, 124.628, 232.264, 72.072, -40.727, 143.741]
  MoveL 1751 to (69.93, 48.83, -161.09) mm, rotated rx -11.83 ry -17.7 rz 126.62 deg; joints [5.115, -38.239, 124.641, 232.24, 72.083, -40.71, 143.741]
  MoveL 1752 to (70.63, 48.8, -161.84) mm, rotated rx -11.83 ry -17.7 rz 126.62 deg; joints [5.072, -38.21, 124.648, 232.188, 72.103, -40.678, 143.741]
  MoveL 1753 to (71.31, 48.46, -162.77) mm, rotated rx -11.83 ry -17.7 rz 126.62 deg; joints [5.026, -38.16, 124.63, 232.133, 72.12, -40.65, 143.741]
  MoveL 1754 to (72.61, 46.85, -165.12) mm, rotated rx -11.83 ry -17.7 rz 126.62 deg; joints [4.922, -37.997, 124.518, 232.014, 72.146, -40.604, 143.741]
  MoveL 1755 to (73.48, 44.58, -167.47) mm, rotated rx -11.83 ry -17.7 rz 126.62 deg; joints [4.832, -37.799, 124.346, 231.917, 72.158, -40.579, 143.741]
  MoveL 1756 to (73.55, 42.24, -169.15) mm, rotated rx -11.83 ry -17.7 rz 126.62 deg; joints [4.787, -37.62, 124.158, 231.874, 72.15, -40.584, 143.741]
  MoveL 1757 to (73.28, 41.04, -169.74) mm, rotated rx -11.83 ry -17.7 rz 126.62 deg; joints [4.781, -37.536, 124.058, 231.873, 72.139, -40.598, 143.741]
  MoveL 1758 to (72.81, 39.83, -170.16) mm, rotated rx -11.83 ry -17.7 rz 126.62 deg; joints [4.787, -37.458, 123.953, 231.884, 72.124, -40.62, 143.741]
  MoveL 1759 to (71.29, 37.34, -170.49) mm, rotated rx -11.83 ry -17.7 rz 126.62 deg; joints [4.83, -37.313, 123.732, 231.948, 72.079, -40.685, 143.741]
  MoveL 1760 to (69.38, 34.84, -170.49) mm, rotated rx -11.83 ry -17.7 rz 126.62 deg; joints [4.895, -37.179, 123.505, 232.038, 72.025, -40.765, 143.741]
  MoveL 1761 to (68.82, 34.03, -170.54) mm, rotated rx -11.83 ry -17.7 rz 126.62 deg; joints [4.913, -37.134, 123.432, 232.063, 72.008, -40.789, 143.741]
  MoveL 1762 to (68.5, 33.62, -170.54) mm, rotated rx -11.83 ry -17.7 rz 126.62 deg; joints [4.924, -37.112, 123.394, 232.077, 71.999, -40.802, 143.741]
  MoveL 1763 to (68.18, 33.19, -170.55) mm, rotated rx -11.83 ry -17.7 rz 126.62 deg; joints [4.935, -37.089, 123.355, 232.093, 71.99, -40.816, 143.741]
  MoveL 1764 to (67.84, 32.73, -170.57) mm, rotated rx -11.83 ry -17.7 rz 126.62 deg; joints [4.946, -37.063, 123.313, 232.108, 71.981, -40.83, 143.741]
  MoveL 1765 to (67.48, 32.19, -170.63) mm, rotated rx -11.83 ry -17.7 rz 126.62 deg; joints [4.957, -37.032, 123.265, 232.123, 71.971, -40.844, 143.741]
  MoveL 1766 to (67.14, 31.72, -170.66) mm, rotated rx -11.83 ry -17.7 rz 126.62 deg; joints [4.967, -37.005, 123.222, 232.138, 71.961, -40.858, 143.741]
  MoveL 1767 to (66.83, 31.3, -170.67) mm, rotated rx -11.83 ry -17.7 rz 126.62 deg; joints [4.977, -36.982, 123.183, 232.152, 71.952, -40.871, 143.741]
  MoveL 1768 to (66.56, 30.9, -170.7) mm, rotated rx -11.83 ry -17.7 rz 126.62 deg; joints [4.986, -36.96, 123.148, 232.164, 71.945, -40.883, 143.741]
  MoveL 1769 to (66.32, 30.52, -170.75) mm, rotated rx -11.83 ry -17.7 rz 126.62 deg; joints [4.993, -36.937, 123.113, 232.175, 71.938, -40.893, 143.741]
  MoveL 1770 to (66.06, 30.14, -170.79) mm, rotated rx -11.83 ry -17.7 rz 126.62 deg; joints [5.001, -36.916, 123.079, 232.186, 71.93, -40.904, 143.741]
  MoveL 1771 to (65.76, 29.73, -170.8) mm, rotated rx -11.83 ry -17.7 rz 126.62 deg; joints [5.011, -36.893, 123.042, 232.2, 71.922, -40.917, 143.741]
  MoveL 1772 to (65.46, 29.32, -170.81) mm, rotated rx -11.83 ry -17.7 rz 126.62 deg; joints [5.02, -36.871, 123.004, 232.213, 71.913, -40.93, 143.741]
  MoveL 1773 to (65.17, 28.88, -170.81) mm, rotated rx -11.83 ry -17.7 rz 126.62 deg; joints [5.03, -36.848, 122.965, 232.227, 71.903, -40.944, 143.741]
  MoveL 1774 to (64.95, 28.45, -170.83) mm, rotated rx -11.83 ry -17.7 rz 126.62 deg; joints [5.036, -36.827, 122.927, 232.237, 71.894, -40.958, 143.741]
  MoveL 1775 to (64.78, 28, -170.86) mm, rotated rx -11.83 ry -17.7 rz 126.62 deg; joints [5.039, -36.805, 122.889, 232.245, 71.883, -40.972, 143.741]
  MoveL 1776 to (64.69, 27.56, -170.91) mm, rotated rx -11.83 ry -17.7 rz 126.62 deg; joints [5.039, -36.785, 122.851, 232.249, 71.873, -40.986, 143.741]
  MoveL 1777 to (64.63, 27.11, -170.95) mm, rotated rx -11.83 ry -17.7 rz 126.62 deg; joints [5.038, -36.765, 122.814, 232.253, 71.862, -41.001, 143.741]
  MoveL 1778 to (65.09, 28.56, -171.92) mm, rotated rx -11.83 ry -17.7 rz 126.62 deg; joints [5.015, -36.769, 122.936, 232.199, 71.933, -40.902, 143.741]
  MoveL 1779 to (65.15, 26.84, -172.3) mm, rotated rx -11.83 ry -17.7 rz 126.62 deg; joints [4.994, -36.689, 122.798, 232.193, 71.896, -40.949, 143.741]
  MoveL 1780 to (65.16, 25.03, -172.58) mm, rotated rx -11.83 ry -17.7 rz 126.62 deg; joints [4.976, -36.611, 122.652, 232.192, 71.854, -41.005, 143.741]
  MoveL 1781 to (65.12, 23.08, -172.78) mm, rotated rx -11.83 ry -17.7 rz 126.62 deg; joints [4.96, -36.531, 122.494, 232.196, 71.805, -41.069, 143.741]
  MoveL 1782 to (65.03, 20.95, -173) mm, rotated rx -11.83 ry -17.7 rz 126.62 deg; joints [4.944, -36.442, 122.32, 232.203, 71.752, -41.139, 143.741]
  MoveL 1783 to (64.92, 18.82, -173.12) mm, rotated rx -11.83 ry -17.7 rz 126.62 deg; joints [4.931, -36.359, 122.146, 232.213, 71.696, -41.214, 143.741]
  MoveL 1784 to (64.81, 16.68, -173.23) mm, rotated rx -11.83 ry -17.7 rz 126.62 deg; joints [4.919, -36.276, 121.972, 232.224, 71.639, -41.289, 143.741]
  MoveL 1785 to (64.71, 14.55, -173.46) mm, rotated rx -11.83 ry -17.7 rz 126.62 deg; joints [4.904, -36.186, 121.798, 232.231, 71.587, -41.359, 143.741]
  MoveL 1786 to (64.6, 12.42, -173.58) mm, rotated rx -11.83 ry -17.7 rz 126.62 deg; joints [4.891, -36.103, 121.623, 232.243, 71.53, -41.434, 143.741]
  MoveL 1787 to (64.47, 10.29, -173.7) mm, rotated rx -11.83 ry -17.7 rz 126.62 deg; joints [4.879, -36.019, 121.448, 232.254, 71.474, -41.509, 143.741]
  MoveL 1788 to (64.36, 8.16, -173.94) mm, rotated rx -11.83 ry -17.7 rz 126.62 deg; joints [4.865, -35.928, 121.273, 232.262, 71.421, -41.579, 143.741]
  MoveL 1789 to (64.23, 6.03, -174.06) mm, rotated rx -11.83 ry -17.7 rz 126.62 deg; joints [4.853, -35.844, 121.098, 232.274, 71.365, -41.654, 143.741]
  MoveL 1790 to (64.1, 3.9, -174.18) mm, rotated rx -11.83 ry -17.7 rz 126.62 deg; joints [4.841, -35.759, 120.922, 232.287, 71.308, -41.729, 143.741]
  MoveL 1791 to (63.97, 1.88, -174.37) mm, rotated rx -11.83 ry -17.7 rz 126.62 deg; joints [4.829, -35.675, 120.756, 232.297, 71.258, -41.797, 143.741]
  MoveL 1792 to (63.85, 0.06, -174.58) mm, rotated rx -11.83 ry -17.7 rz 126.62 deg; joints [4.818, -35.595, 120.606, 232.304, 71.213, -41.856, 143.741]
  MoveL 1793 to (63.73, -1.9, -174.69) mm, rotated rx -11.83 ry -17.7 rz 126.62 deg; joints [4.808, -35.518, 120.444, 232.316, 71.161, -41.925, 143.741]
  MoveL 1794 to (63.69, -4.07, -174.69) mm, rotated rx -11.83 ry -17.7 rz 126.62 deg; joints [4.793, -35.44, 120.266, 232.329, 71.098, -42.009, 143.741]
  MoveL 1795 to (63.5, -6.78, -174.78) mm, rotated rx -11.83 ry -17.7 rz 126.62 deg; joints [4.781, -35.335, 120.041, 232.349, 71.024, -42.108, 143.741]
  MoveL 1796 to (63.22, -9.23, -175.02) mm, rotated rx -11.83 ry -17.7 rz 126.62 deg; joints [4.772, -35.228, 119.836, 232.366, 70.964, -42.19, 143.741]
  MoveL 1797 to (63.07, -11.26, -175.2) mm, rotated rx -11.83 ry -17.7 rz 126.62 deg; joints [4.761, -35.143, 119.667, 232.378, 70.912, -42.259, 143.741]
  MoveL 1798 to (62.91, -13.12, -175.52) mm, rotated rx -11.83 ry -17.7 rz 126.62 deg; joints [4.749, -35.055, 119.511, 232.385, 70.87, -42.315, 143.741]
  MoveL 1799 to (62.76, -15.16, -175.7) mm, rotated rx -11.83 ry -17.7 rz 126.62 deg; joints [4.739, -34.968, 119.341, 232.398, 70.818, -42.385, 143.741]
  MoveL 1800 to (62.59, -17.13, -175.9) mm, rotated rx -11.83 ry -17.7 rz 126.62 deg; joints [4.729, -34.883, 119.176, 232.41, 70.769, -42.451, 143.741]
  MoveL 1801 to (62.39, -19.05, -176.18) mm, rotated rx -11.83 ry -17.7 rz 126.62 deg; joints [4.72, -34.794, 119.015, 232.42, 70.724, -42.511, 143.741]
  MoveL 1802 to (61.8, -19.74, -176.95) mm, rotated rx -11.83 ry -17.7 rz 126.62 deg; joints [4.729, -34.712, 118.948, 232.426, 70.734, -42.499, 143.741]
  MoveL 1803 to (61.63, -19.4, -177.33) mm, rotated rx -11.83 ry -17.7 rz 126.62 deg; joints [4.733, -34.698, 118.972, 232.419, 70.758, -42.467, 143.741]
  MoveL 1804 to (61.57, -19.35, -177.57) mm, rotated rx -11.83 ry -17.7 rz 126.62 deg; joints [4.733, -34.685, 118.976, 232.414, 70.768, -42.453, 143.741]
  MoveL 1805 to (61.63, -19.55, -177.7) mm, rotated rx -11.83 ry -17.7 rz 126.62 deg; joints [4.728, -34.671, 118.959, 232.41, 70.765, -42.455, 143.741]
  MoveL 1806 to (61.84, -20.03, -177.75) mm, rotated rx -11.83 ry -17.7 rz 126.62 deg; joints [4.715, -34.657, 118.923, 232.402, 70.751, -42.473, 143.741]
  MoveL 1807 to (62.14, -20.63, -177.79) mm, rotated rx -11.83 ry -17.7 rz 126.62 deg; joints [4.697, -34.641, 118.878, 232.393, 70.732, -42.496, 143.741]
  MoveL 1808 to (62.93, -21.99, -177.79) mm, rotated rx -11.83 ry -17.7 rz 126.62 deg; joints [4.654, -34.612, 118.778, 232.369, 70.685, -42.554, 143.741]
  MoveL 1809 to (63.2, -22.46, -177.79) mm, rotated rx -11.83 ry -17.7 rz 126.62 deg; joints [4.639, -34.602, 118.742, 232.361, 70.668, -42.573, 143.741]
  MoveL 1810 to (63.45, -22.93, -177.82) mm, rotated rx -11.83 ry -17.7 rz 126.62 deg; joints [4.625, -34.59, 118.707, 232.353, 70.653, -42.592, 143.741]
  MoveL 1811 to (63.7, -23.42, -177.87) mm, rotated rx -11.83 ry -17.7 rz 126.62 deg; joints [4.611, -34.576, 118.67, 232.344, 70.638, -42.61, 143.741]
  MoveL 1812 to (63.94, -23.93, -177.94) mm, rotated rx -11.83 ry -17.7 rz 126.62 deg; joints [4.596, -34.559, 118.631, 232.336, 70.623, -42.628, 143.741]
  MoveL 1813 to (64.18, -24.42, -178) mm, rotated rx -11.83 ry -17.7 rz 126.62 deg; joints [4.582, -34.544, 118.594, 232.328, 70.608, -42.646, 143.741]
  MoveL 1814 to (64.42, -24.86, -178.02) mm, rotated rx -11.83 ry -17.7 rz 126.62 deg; joints [4.568, -34.533, 118.561, 232.32, 70.594, -42.663, 143.741]
  MoveL 1815 to (64.64, -25.26, -178.04) mm, rotated rx -11.83 ry -17.7 rz 126.62 deg; joints [4.556, -34.524, 118.531, 232.313, 70.58, -42.679, 143.741]
  MoveL 1816 to (65.43, -26.62, -178.04) mm, rotated rx -11.83 ry -17.7 rz 126.62 deg; joints [4.513, -34.495, 118.43, 232.29, 70.533, -42.737, 143.741]
  MoveL 1817 to (65.68, -27.07, -178.05) mm, rotated rx -11.83 ry -17.7 rz 126.62 deg; joints [4.499, -34.484, 118.396, 232.282, 70.517, -42.755, 143.741]
  MoveL 1818 to (65.9, -27.49, -178.08) mm, rotated rx -11.83 ry -17.7 rz 126.62 deg; joints [4.487, -34.473, 118.365, 232.275, 70.504, -42.771, 143.741]
  MoveL 1819 to (66.09, -27.9, -178.13) mm, rotated rx -11.83 ry -17.7 rz 126.62 deg; joints [4.475, -34.46, 118.334, 232.268, 70.492, -42.786, 143.741]
  MoveL 1820 to (66.3, -28.3, -178.17) mm, rotated rx -11.83 ry -17.7 rz 126.62 deg; joints [4.463, -34.449, 118.303, 232.262, 70.479, -42.801, 143.741]
  MoveL 1821 to (66.54, -28.73, -178.18) mm, rotated rx -11.83 ry -17.7 rz 126.62 deg; joints [4.45, -34.439, 118.271, 232.255, 70.465, -42.819, 143.741]
  MoveL 1822 to (66.8, -29.18, -178.18) mm, rotated rx -11.83 ry -17.7 rz 126.62 deg; joints [4.436, -34.429, 118.238, 232.247, 70.449, -42.838, 143.741]
  MoveL 1823 to (68.01, -31.85, -178.52) mm, rotated rx -11.83 ry -17.7 rz 126.62 deg; joints [4.362, -34.344, 118.033, 232.206, 70.369, -42.933, 143.741]
  MoveL 1824 to (68.33, -33.12, -178.94) mm, rotated rx -11.83 ry -17.7 rz 126.62 deg; joints [4.335, -34.282, 117.931, 232.189, 70.342, -42.965, 143.741]
  MoveL 1825 to (68.46, -34.36, -179.53) mm, rotated rx -11.83 ry -17.7 rz 126.62 deg; joints [4.313, -34.208, 117.829, 232.174, 70.323, -42.987, 143.741]
  MoveL 1826 to (68.14, -36.73, -181.22) mm, rotated rx -11.83 ry -17.7 rz 126.62 deg; joints [4.287, -34.021, 117.624, 232.153, 70.309, -43, 143.741]
  MoveL 1827 to (67.05, -38.94, -183.58) mm, rotated rx -11.83 ry -17.7 rz 126.62 deg; joints [4.285, -33.783, 117.419, 232.142, 70.329, -42.973, 143.741]
  MoveL 1828 to (65.6, -40.44, -185.95) mm, rotated rx -11.83 ry -17.7 rz 126.62 deg; joints [4.302, -33.563, 117.267, 232.14, 70.373, -42.916, 143.741]
  MoveL 1829 to (64.9, -40.72, -186.87) mm, rotated rx -11.83 ry -17.7 rz 126.62 deg; joints [4.317, -33.484, 117.231, 232.143, 70.401, -42.881, 143.741]
  MoveL 1830 to (64.21, -40.68, -187.63) mm, rotated rx -11.83 ry -17.7 rz 126.62 deg; joints [4.335, -33.426, 117.222, 232.148, 70.432, -42.841, 143.741]
  MoveL 1831 to (63.88, -40.54, -187.95) mm, rotated rx -11.83 ry -17.7 rz 126.62 deg; joints [4.346, -33.405, 117.228, 232.151, 70.449, -42.82, 143.741]
  MoveL 1832 to (63.54, -40.32, -188.22) mm, rotated rx -11.83 ry -17.7 rz 126.62 deg; joints [4.357, -33.39, 117.24, 232.155, 70.468, -42.797, 143.741]
  MoveL 1833 to (62.89, -39.65, -188.65) mm, rotated rx -11.83 ry -17.7 rz 126.62 deg; joints [4.383, -33.374, 117.286, 232.164, 70.507, -42.748, 143.741]
  MoveL 1834 to (62.25, -38.66, -188.9) mm, rotated rx -11.83 ry -17.7 rz 126.62 deg; joints [4.413, -33.379, 117.358, 232.176, 70.551, -42.694, 143.741]
  MoveL 1835 to (61.62, -37.36, -188.98) mm, rotated rx -11.83 ry -17.7 rz 126.62 deg; joints [4.447, -33.405, 117.457, 232.19, 70.598, -42.635, 143.741]
  MoveL 1836 to (61.01, -35.91, -188.98) mm, rotated rx -11.83 ry -17.7 rz 126.62 deg; joints [4.482, -33.441, 117.568, 232.205, 70.647, -42.574, 143.741]
  MoveL 1837 to (60.81, -35.42, -188.98) mm, rotated rx -11.83 ry -17.7 rz 126.62 deg; joints [4.494, -33.454, 117.606, 232.21, 70.664, -42.554, 143.741]
  MoveL 1838 to (60.61, -34.88, -188.94) mm, rotated rx -11.83 ry -17.7 rz 126.62 deg; joints [4.507, -33.47, 117.648, 232.216, 70.681, -42.533, 143.741]
  MoveL 1839 to (60.4, -34.27, -188.88) mm, rotated rx -11.83 ry -17.7 rz 126.62 deg; joints [4.52, -33.49, 117.696, 232.222, 70.699, -42.511, 143.741]
  MoveL 1840 to (60.2, -33.74, -188.85) mm, rotated rx -11.83 ry -17.7 rz 126.62 deg; joints [4.533, -33.505, 117.737, 232.228, 70.715, -42.49, 143.741]
  MoveL 1841 to (60, -33.25, -188.85) mm, rotated rx -11.83 ry -17.7 rz 126.62 deg; joints [4.545, -33.518, 117.774, 232.233, 70.732, -42.47, 143.741]
  MoveL 1842 to (59.8, -32.77, -188.84) mm, rotated rx -11.83 ry -17.7 rz 126.62 deg; joints [4.557, -33.53, 117.811, 232.238, 70.748, -42.45, 143.741]
  MoveL 1843 to (59.63, -32.29, -188.79) mm, rotated rx -11.83 ry -17.7 rz 126.62 deg; joints [4.568, -33.546, 117.849, 232.243, 70.762, -42.432, 143.741]
  MoveL 1844 to (59.49, -31.81, -188.72) mm, rotated rx -11.83 ry -17.7 rz 126.62 deg; joints [4.578, -33.564, 117.887, 232.248, 70.775, -42.416, 143.741]
  MoveL 1845 to (59.35, -31.32, -188.62) mm, rotated rx -11.83 ry -17.7 rz 126.62 deg; joints [4.589, -33.583, 117.925, 232.253, 70.788, -42.4, 143.741]
  MoveL 1846 to (59.2, -30.84, -188.55) mm, rotated rx -11.83 ry -17.7 rz 126.62 deg; joints [4.599, -33.6, 117.964, 232.258, 70.802, -42.384, 143.741]
  MoveL 1847 to (59.01, -30.34, -188.52) mm, rotated rx -11.83 ry -17.7 rz 126.62 deg; joints [4.611, -33.615, 118.002, 232.264, 70.817, -42.364, 143.741]
  MoveL 1848 to (58.81, -29.86, -188.51) mm, rotated rx -11.83 ry -17.7 rz 126.62 deg; joints [4.623, -33.628, 118.039, 232.269, 70.833, -42.345, 143.741]
  MoveL 1849 to (57.86, -27.49, -188.5) mm, rotated rx -11.83 ry -17.7 rz 126.62 deg; joints [4.68, -33.687, 118.221, 232.293, 70.912, -42.246, 143.741]
  MoveL 1850 to (57.76, -27.11, -188.48) mm, rotated rx -11.83 ry -17.7 rz 126.62 deg; joints [4.687, -33.7, 118.251, 232.296, 70.923, -42.232, 143.741]
  MoveL 1851 to (57.75, -26.94, -188.36) mm, rotated rx -11.83 ry -17.7 rz 126.62 deg; joints [4.69, -33.712, 118.265, 232.298, 70.925, -42.23, 143.741]
  MoveL 1852 to (57.77, -27.03, -188.13) mm, rotated rx -11.83 ry -17.7 rz 126.62 deg; joints [4.692, -33.722, 118.259, 232.305, 70.915, -42.244, 143.741]
  MoveL 1853 to (57.82, -27.38, -187.77) mm, rotated rx -11.83 ry -17.7 rz 126.62 deg; joints [4.692, -33.732, 118.231, 232.315, 70.892, -42.275, 143.741]
  MoveL 1854 to (58.36, -26.83, -187.03) mm, rotated rx -11.83 ry -17.7 rz 126.62 deg; joints [4.684, -33.806, 118.287, 232.312, 70.88, -42.29, 143.741]
  MoveL 1855 to (58.76, -24.75, -187.01) mm, rotated rx -11.83 ry -17.7 rz 126.62 deg; joints [4.682, -33.89, 118.465, 232.284, 70.938, -42.211, 143.741]
  MoveL 1856 to (59.21, -22.61, -186.88) mm, rotated rx -11.83 ry -17.7 rz 126.62 deg; joints [4.68, -33.983, 118.649, 232.257, 70.993, -42.136, 143.741]
  MoveL 1857 to (59.71, -20.39, -186.62) mm, rotated rx -11.83 ry -17.7 rz 126.62 deg; joints [4.678, -34.088, 118.84, 232.232, 71.045, -42.063, 143.741]
  MoveL 1858 to (60.15, -18.32, -186.49) mm, rotated rx -11.83 ry -17.7 rz 126.62 deg; joints [4.676, -34.178, 119.017, 232.207, 71.098, -41.991, 143.741]
  MoveL 1859 to (60.58, -16.32, -186.23) mm, rotated rx -11.83 ry -17.7 rz 126.62 deg; joints [4.676, -34.273, 119.189, 232.186, 71.145, -41.927, 143.741]
  MoveL 1860 to (61.03, -14.27, -185.87) mm, rotated rx -11.83 ry -17.7 rz 126.62 deg; joints [4.676, -34.376, 119.366, 232.166, 71.191, -41.865, 143.741]
  MoveL 1861 to (61.46, -12.16, -185.73) mm, rotated rx -11.83 ry -17.7 rz 126.62 deg; joints [4.675, -34.468, 119.545, 232.142, 71.244, -41.792, 143.741]
  MoveL 1862 to (61.87, -10.09, -185.63) mm, rotated rx -11.83 ry -17.7 rz 126.62 deg; joints [4.674, -34.556, 119.721, 232.117, 71.299, -41.718, 143.741]
  MoveL 1863 to (62.28, -7.98, -185.49) mm, rotated rx -11.83 ry -17.7 rz 126.62 deg; joints [4.673, -34.647, 119.9, 232.093, 71.352, -41.645, 143.741]
  MoveL 1864 to (62.72, -5.94, -185.2) mm, rotated rx -11.83 ry -17.7 rz 126.62 deg; joints [4.673, -34.746, 120.075, 232.073, 71.399, -41.582, 143.741]
  MoveL 1865 to (63.1, -3.78, -184.86) mm, rotated rx -11.83 ry -17.7 rz 126.62 deg; joints [4.678, -34.849, 120.257, 232.056, 71.448, -41.516, 143.741]
  MoveL 1866 to (63.49, -1.7, -184.68) mm, rotated rx -11.83 ry -17.7 rz 126.62 deg; joints [4.678, -34.941, 120.434, 232.034, 71.5, -41.446, 143.741]
  MoveL 1867 to (63.89, 0.41, -184.57) mm, rotated rx -11.83 ry -17.7 rz 126.62 deg; joints [4.678, -35.03, 120.612, 232.01, 71.555, -41.372, 143.741]
  MoveL 1868 to (64.29, 2.5, -184.5) mm, rotated rx -11.83 ry -17.7 rz 126.62 deg; joints [4.677, -35.116, 120.788, 231.986, 71.61, -41.297, 143.741]
  MoveL 1869 to (64.67, 4.6, -184.27) mm, rotated rx -11.83 ry -17.7 rz 126.62 deg; joints [4.679, -35.21, 120.966, 231.966, 71.662, -41.228, 143.741]
  MoveL 1870 to (65.05, 6.69, -184.14) mm, rotated rx -11.83 ry -17.7 rz 126.62 deg; joints [4.68, -35.3, 121.141, 231.944, 71.715, -41.156, 143.741]
  MoveL 1871 to (65.45, 8.8, -184.06) mm, rotated rx -11.83 ry -17.7 rz 126.62 deg; joints [4.679, -35.386, 121.318, 231.92, 71.771, -41.081, 143.741]
  MoveL 1872 to (65.8, 10.89, -183.83) mm, rotated rx -11.83 ry -17.7 rz 126.62 deg; joints [4.682, -35.48, 121.494, 231.902, 71.822, -41.013, 143.741]
  MoveL 1873 to (66.16, 13.02, -183.6) mm, rotated rx -11.83 ry -17.7 rz 126.62 deg; joints [4.685, -35.575, 121.672, 231.884, 71.873, -40.945, 143.741]
  MoveL 1874 to (66.54, 15.16, -183.45) mm, rotated rx -11.83 ry -17.7 rz 126.62 deg; joints [4.687, -35.666, 121.851, 231.863, 71.927, -40.872, 143.741]
  MoveL 1875 to (66.83, 17.02, -183.32) mm, rotated rx -11.83 ry -17.7 rz 126.62 deg; joints [4.69, -35.744, 122.006, 231.846, 71.975, -40.809, 143.741]
  MoveL 1876 to (67.03, 18.65, -183.11) mm, rotated rx -11.83 ry -17.7 rz 126.62 deg; joints [4.696, -35.817, 122.141, 231.836, 72.014, -40.757, 143.741]
  MoveL 1877 to (67.12, 20.08, -182.79) mm, rotated rx -11.83 ry -17.7 rz 126.62 deg; joints [4.707, -35.887, 122.259, 231.835, 72.044, -40.718, 143.741]
  MoveL 1878 to (66.63, 18.69, -181.83) mm, rotated rx -11.83 ry -17.7 rz 126.62 deg; joints [4.732, -35.884, 122.142, 231.889, 71.975, -40.813, 143.741]
  MoveL 1879 to (66.72, 19.18, -181.83) mm, rotated rx -11.83 ry -17.7 rz 126.62 deg; joints [4.731, -35.903, 122.183, 231.883, 71.988, -40.795, 143.741]
  MoveL 1880 to (66.86, 19.66, -181.83) mm, rotated rx -11.83 ry -17.7 rz 126.62 deg; joints [4.729, -35.923, 122.224, 231.876, 72.001, -40.778, 143.741]
  MoveL 1881 to (67.09, 20.14, -181.8) mm, rotated rx -11.83 ry -17.7 rz 126.62 deg; joints [4.723, -35.946, 122.266, 231.865, 72.012, -40.763, 143.741]
  MoveL 1882 to (67.39, 20.61, -181.76) mm, rotated rx -11.83 ry -17.7 rz 126.62 deg; joints [4.714, -35.972, 122.308, 231.851, 72.022, -40.749, 143.741]
  MoveL 1883 to (67.76, 21.1, -181.71) mm, rotated rx -11.83 ry -17.7 rz 126.62 deg; joints [4.702, -36.002, 122.353, 231.836, 72.031, -40.735, 143.741]
  MoveL 1884 to (68.15, 21.53, -181.67) mm, rotated rx -11.83 ry -17.7 rz 126.62 deg; joints [4.689, -36.028, 122.394, 231.819, 72.039, -40.723, 143.741]
  MoveL 1885 to (68.54, 21.94, -181.65) mm, rotated rx -11.83 ry -17.7 rz 126.62 deg; joints [4.675, -36.053, 122.432, 231.801, 72.047, -40.711, 143.741]
  MoveL 1886 to (68.9, 22.31, -181.65) mm, rotated rx -11.83 ry -17.7 rz 126.62 deg; joints [4.662, -36.075, 122.468, 231.785, 72.054, -40.7, 143.741]
  MoveL 1887 to (69.27, 22.69, -181.65) mm, rotated rx -11.83 ry -17.7 rz 126.62 deg; joints [4.649, -36.098, 122.504, 231.768, 72.062, -40.688, 143.741]
  MoveL 1888 to (69.66, 23.13, -181.6) mm, rotated rx -11.83 ry -17.7 rz 126.62 deg; joints [4.636, -36.125, 122.545, 231.751, 72.07, -40.676, 143.741]
  MoveL 1889 to (70.08, 23.64, -181.52) mm, rotated rx -11.83 ry -17.7 rz 126.62 deg; joints [4.622, -36.158, 122.592, 231.734, 72.078, -40.664, 143.741]
  MoveL 1890 to (70.42, 24.03, -181.47) mm, rotated rx -11.83 ry -17.7 rz 126.62 deg; joints [4.611, -36.183, 122.628, 231.719, 72.085, -40.654, 143.741]
  MoveL 1891 to (70.71, 24.34, -181.44) mm, rotated rx -11.83 ry -17.7 rz 126.62 deg; joints [4.601, -36.202, 122.658, 231.707, 72.09, -40.645, 143.741]
  MoveL 1892 to (71.05, 24.69, -181.43) mm, rotated rx -11.83 ry -17.7 rz 126.62 deg; joints [4.589, -36.223, 122.69, 231.692, 72.097, -40.635, 143.741]
  MoveL 1893 to (71.41, 25.06, -181.43) mm, rotated rx -11.83 ry -17.7 rz 126.62 deg; joints [4.576, -36.245, 122.725, 231.675, 72.104, -40.624, 143.741]
  MoveL 1894 to (71.76, 25.43, -181.41) mm, rotated rx -11.83 ry -17.7 rz 126.62 deg; joints [4.564, -36.267, 122.76, 231.66, 72.112, -40.613, 143.741]
  MoveL 1895 to (72.1, 25.79, -181.39) mm, rotated rx -11.83 ry -17.7 rz 126.62 deg; joints [4.552, -36.29, 122.795, 231.645, 72.118, -40.603, 143.741]
  MoveL 1896 to (72.45, 26.16, -181.38) mm, rotated rx -11.83 ry -17.7 rz 126.62 deg; joints [4.539, -36.312, 122.829, 231.629, 72.126, -40.592, 143.741]
  MoveL 1897 to (74.3, 28.03, -181.37) mm, rotated rx -11.83 ry -17.7 rz 126.62 deg; joints [4.472, -36.422, 123.006, 231.544, 72.163, -40.535, 143.741]
  MoveL 1898 to (75.37, 29.01, -181.46) mm, rotated rx -11.83 ry -17.7 rz 126.62 deg; joints [4.431, -36.478, 123.1, 231.493, 72.186, -40.502, 143.741]
  MoveL 1899 to (76.34, 29.72, -181.71) mm, rotated rx -11.83 ry -17.7 rz 126.62 deg; joints [4.39, -36.511, 123.169, 231.442, 72.206, -40.47, 143.741]
  MoveL 1900 to (77.22, 30.14, -182.12) mm, rotated rx -11.83 ry -17.7 rz 126.62 deg; joints [4.348, -36.523, 123.214, 231.392, 72.225, -40.441, 143.741]
  MoveL 1901 to (77.99, 30.27, -182.71) mm, rotated rx -11.83 ry -17.7 rz 126.62 deg; joints [4.307, -36.512, 123.234, 231.343, 72.242, -40.415, 143.741]
  MoveL 1902 to (78.67, 30.13, -183.46) mm, rotated rx -11.83 ry -17.7 rz 126.62 deg; joints [4.265, -36.479, 123.23, 231.293, 72.258, -40.39, 143.741]
  MoveL 1903 to (79.25, 29.69, -184.37) mm, rotated rx -11.83 ry -17.7 rz 126.62 deg; joints [4.223, -36.424, 123.201, 231.245, 72.273, -40.367, 143.741]
  MoveL 1904 to (80.11, 27.98, -186.7) mm, rotated rx -11.83 ry -17.7 rz 126.62 deg; joints [4.139, -36.249, 123.068, 231.149, 72.296, -40.329, 143.741]
  MoveL 1905 to (80.41, 25.73, -189.05) mm, rotated rx -11.83 ry -17.7 rz 126.62 deg; joints [4.077, -36.04, 122.884, 231.08, 72.309, -40.306, 143.741]
  MoveL 1906 to (79.94, 23.51, -190.76) mm, rotated rx -11.83 ry -17.7 rz 126.62 deg; joints [4.057, -35.852, 122.693, 231.06, 72.306, -40.308, 143.741]
  MoveL 1907 to (79.43, 22.41, -191.37) mm, rotated rx -11.83 ry -17.7 rz 126.62 deg; joints [4.063, -35.765, 122.596, 231.069, 72.3, -40.317, 143.741]
  MoveL 1908 to (78.72, 21.32, -191.82) mm, rotated rx -11.83 ry -17.7 rz 126.62 deg; joints [4.08, -35.684, 122.497, 231.09, 72.289, -40.332, 143.741]
  MoveL 1909 to (76.75, 19.18, -192.25) mm, rotated rx -11.83 ry -17.7 rz 126.62 deg; joints [4.145, -35.537, 122.295, 231.17, 72.258, -40.379, 143.741]
  MoveL 1910 to (76, 18.5, -192.29) mm, rotated rx -11.83 ry -17.7 rz 126.62 deg; joints [4.172, -35.493, 122.23, 231.203, 72.246, -40.398, 143.741]
  MoveL 1911 to (73.93, 16.89, -192.29) mm, rotated rx -11.83 ry -17.7 rz 126.62 deg; joints [4.251, -35.387, 122.071, 231.296, 72.216, -40.444, 143.741]
  MoveL 1912 to (73.16, 16.24, -192.35) mm, rotated rx -11.83 ry -17.7 rz 126.62 deg; joints [4.279, -35.343, 122.007, 231.329, 72.205, -40.461, 143.741]
  MoveL 1913 to (72.33, 15.59, -192.35) mm, rotated rx -11.83 ry -17.7 rz 126.62 deg; joints [4.31, -35.3, 121.943, 231.366, 72.193, -40.48, 143.741]
  MoveL 1914 to (71.96, 15.29, -192.36) mm, rotated rx -11.83 ry -17.7 rz 126.62 deg; joints [4.325, -35.28, 121.913, 231.383, 72.188, -40.488, 143.741]
  MoveL 1915 to (71.63, 15.01, -192.38) mm, rotated rx -11.83 ry -17.7 rz 126.62 deg; joints [4.336, -35.261, 121.886, 231.397, 72.183, -40.496, 143.741]
  MoveL 1916 to (71.27, 14.72, -192.39) mm, rotated rx -11.83 ry -17.7 rz 126.62 deg; joints [4.35, -35.241, 121.857, 231.413, 72.178, -40.504, 143.741]
  MoveL 1917 to (69.21, 13.11, -192.4) mm, rotated rx -11.83 ry -17.7 rz 126.62 deg; joints [4.428, -35.135, 121.697, 231.505, 72.148, -40.551, 143.741]
  MoveL 1918 to (68.83, 12.79, -192.42) mm, rotated rx -11.83 ry -17.7 rz 126.62 deg; joints [4.442, -35.114, 121.666, 231.522, 72.142, -40.56, 143.741]
  MoveL 1919 to (68.49, 12.48, -192.45) mm, rotated rx -11.83 ry -17.7 rz 126.62 deg; joints [4.454, -35.093, 121.635, 231.536, 72.137, -40.568, 143.741]
  MoveL 1920 to (68.19, 12.16, -192.49) mm, rotated rx -11.83 ry -17.7 rz 126.62 deg; joints [4.464, -35.072, 121.605, 231.549, 72.132, -40.576, 143.741]
  MoveL 1921 to (67.92, 11.81, -192.53) mm, rotated rx -11.83 ry -17.7 rz 126.62 deg; joints [4.473, -35.052, 121.573, 231.56, 72.125, -40.586, 143.741]
  MoveL 1922 to (67.7, 11.43, -192.55) mm, rotated rx -11.83 ry -17.7 rz 126.62 deg; joints [4.479, -35.032, 121.539, 231.571, 72.116, -40.598, 143.741]
  MoveL 1923 to (67.52, 11.02, -192.55) mm, rotated rx -11.83 ry -17.7 rz 126.62 deg; joints [4.484, -35.014, 121.503, 231.58, 72.106, -40.613, 143.741]
  MoveL 1924 to (67.95, 11.65, -193.29) mm, rotated rx -11.83 ry -17.7 rz 126.62 deg; joints [4.459, -35.002, 121.558, 231.538, 72.146, -40.557, 143.741]
  MoveL 1925 to (67.75, 10.24, -193.84) mm, rotated rx -11.83 ry -17.7 rz 126.62 deg; joints [4.45, -34.917, 121.438, 231.538, 72.124, -40.585, 143.741]
  MoveL 1926 to (67.43, 8.71, -194.27) mm, rotated rx -11.83 ry -17.7 rz 126.62 deg; joints [4.447, -34.833, 121.308, 231.546, 72.095, -40.623, 143.741]
  MoveL 1927 to (66.99, 6.99, -194.57) mm, rotated rx -11.83 ry -17.7 rz 126.62 deg; joints [4.449, -34.746, 121.161, 231.564, 72.058, -40.672, 143.741]
  MoveL 1928 to (66.4, 5.06, -194.76) mm, rotated rx -11.83 ry -17.7 rz 126.62 deg; joints [4.458, -34.655, 120.995, 231.592, 72.011, -40.735, 143.741]
  MoveL 1929 to (65.78, 3.06, -194.95) mm, rotated rx -11.83 ry -17.7 rz 126.62 deg; joints [4.468, -34.561, 120.822, 231.622, 71.963, -40.8, 143.741]
  MoveL 1930 to (65.13, 1.03, -195.07) mm, rotated rx -11.83 ry -17.7 rz 126.62 deg; joints [4.48, -34.47, 120.647, 231.655, 71.912, -40.869, 143.741]
  MoveL 1931 to (64.49, -1.01, -195.3) mm, rotated rx -11.83 ry -17.7 rz 126.62 deg; joints [4.49, -34.371, 120.471, 231.685, 71.864, -40.934, 143.741]
  MoveL 1932 to (63.84, -3.04, -195.41) mm, rotated rx -11.83 ry -17.7 rz 126.62 deg; joints [4.502, -34.28, 120.295, 231.719, 71.813, -41.004, 143.741]
  MoveL 1933 to (63.18, -5.07, -195.53) mm, rotated rx -11.83 ry -17.7 rz 126.62 deg; joints [4.514, -34.188, 120.12, 231.753, 71.761, -41.074, 143.741]
  MoveL 1934 to (62.52, -7.1, -195.65) mm, rotated rx -11.83 ry -17.7 rz 126.62 deg; joints [4.526, -34.096, 119.944, 231.787, 71.71, -41.144, 143.741]
  MoveL 1935 to (61.86, -9.13, -195.88) mm, rotated rx -11.83 ry -17.7 rz 126.62 deg; joints [4.537, -33.997, 119.767, 231.818, 71.663, -41.209, 143.741]
  MoveL 1936 to (61.19, -11.16, -196) mm, rotated rx -11.83 ry -17.7 rz 126.62 deg; joints [4.549, -33.904, 119.59, 231.853, 71.611, -41.279, 143.741]
  MoveL 1937 to (60.61, -13.12, -196.1) mm, rotated rx -11.83 ry -17.7 rz 126.62 deg; joints [4.559, -33.817, 119.42, 231.884, 71.561, -41.348, 143.741]
  MoveL 1938 to (60.15, -15.08, -196.31) mm, rotated rx -11.83 ry -17.7 rz 126.62 deg; joints [4.562, -33.727, 119.252, 231.908, 71.513, -41.413, 143.741]
  MoveL 1939 to (59.34, -17.45, -196.45) mm, rotated rx -11.83 ry -17.7 rz 126.62 deg; joints [4.577, -33.618, 119.044, 231.949, 71.453, -41.496, 143.741]
  MoveL 1940 to (58.43, -19.73, -196.53) mm, rotated rx -11.83 ry -17.7 rz 126.62 deg; joints [4.598, -33.513, 118.843, 231.996, 71.395, -41.577, 143.741]
  MoveL 1941 to (57.64, -21.87, -196.56) mm, rotated rx -11.83 ry -17.7 rz 126.62 deg; joints [4.616, -33.418, 118.655, 232.039, 71.339, -41.656, 143.741]
  MoveL 1942 to (56.98, -23.82, -196.61) mm, rotated rx -11.83 ry -17.7 rz 126.62 deg; joints [4.63, -33.332, 118.484, 232.075, 71.287, -41.727, 143.741]
  MoveL 1943 to (56.36, -25.68, -196.73) mm, rotated rx -11.83 ry -17.7 rz 126.62 deg; joints [4.641, -33.246, 118.321, 232.108, 71.241, -41.792, 143.741]
  MoveL 1944 to (55.72, -27.6, -196.79) mm, rotated rx -11.83 ry -17.7 rz 126.62 deg; joints [4.653, -33.16, 118.152, 232.142, 71.19, -41.862, 143.741]
  MoveL 1945 to (55.05, -29.62, -196.86) mm, rotated rx -11.83 ry -17.7 rz 126.62 deg; joints [4.667, -33.07, 117.975, 232.179, 71.138, -41.935, 143.741]
  MoveL 1946 to (54.39, -31.5, -197.04) mm, rotated rx -11.83 ry -17.7 rz 126.62 deg; joints [4.678, -32.979, 117.809, 232.211, 71.093, -41.999, 143.741]
  MoveL 1947 to (53.74, -33.29, -197.36) mm, rotated rx -11.83 ry -17.7 rz 126.62 deg; joints [4.689, -32.883, 117.649, 232.239, 71.055, -42.052, 143.741]
  MoveL 1948 to (53.08, -33.85, -198.4) mm, rotated rx -11.83 ry -17.7 rz 126.62 deg; joints [4.698, -32.789, 117.589, 232.239, 71.076, -42.024, 143.741]
  MoveL 1949 to (53.11, -33.59, -198.92) mm, rotated rx -11.83 ry -17.7 rz 126.62 deg; joints [4.692, -32.769, 117.608, 232.222, 71.1, -41.991, 143.741]
  MoveL 1950 to (53.09, -33.57, -199.24) mm, rotated rx -11.83 ry -17.7 rz 126.62 deg; joints [4.688, -32.751, 117.608, 232.214, 71.111, -41.976, 143.741]
  MoveL 1951 to (53.04, -33.78, -199.4) mm, rotated rx -11.83 ry -17.7 rz 126.62 deg; joints [4.686, -32.733, 117.59, 232.212, 71.11, -41.977, 143.741]
  MoveL 1952 to (53.01, -34.2, -199.44) mm, rotated rx -11.83 ry -17.7 rz 126.62 deg; joints [4.684, -32.715, 117.554, 232.215, 71.099, -41.992, 143.741]
  MoveL 1953 to (53.02, -34.72, -199.46) mm, rotated rx -11.83 ry -17.7 rz 126.62 deg; joints [4.68, -32.697, 117.511, 232.217, 71.083, -42.012, 143.741]
  MoveL 1954 to (53.12, -35.31, -199.47) mm, rotated rx -11.83 ry -17.7 rz 126.62 deg; joints [4.671, -32.678, 117.464, 232.216, 71.065, -42.035, 143.741]
  MoveL 1955 to (53.26, -35.92, -199.48) mm, rotated rx -11.83 ry -17.7 rz 126.62 deg; joints [4.661, -32.66, 117.415, 232.214, 71.046, -42.06, 143.741]
  MoveL 1956 to (54.24, -39.45, -199.48) mm, rotated rx -11.83 ry -17.7 rz 126.62 deg; joints [4.595, -32.562, 117.136, 232.196, 70.931, -42.207, 143.741]
  MoveL 1957 to (54.35, -39.88, -199.51) mm, rotated rx -11.83 ry -17.7 rz 126.62 deg; joints [4.588, -32.548, 117.102, 232.194, 70.917, -42.223, 143.741]
  MoveL 1958 to (54.47, -40.35, -199.52) mm, rotated rx -11.83 ry -17.7 rz 126.62 deg; joints [4.579, -32.534, 117.065, 232.192, 70.902, -42.242, 143.741]
  MoveL 1959 to (54.61, -40.86, -199.52) mm, rotated rx -11.83 ry -17.7 rz 126.62 deg; joints [4.57, -32.519, 117.025, 232.189, 70.886, -42.263, 143.741]
  MoveL 1960 to (54.73, -41.33, -199.54) mm, rotated rx -11.83 ry -17.7 rz 126.62 deg; joints [4.561, -32.505, 116.987, 232.187, 70.871, -42.282, 143.741]
  MoveL 1961 to (54.83, -41.79, -199.58) mm, rotated rx -11.83 ry -17.7 rz 126.62 deg; joints [4.553, -32.489, 116.95, 232.185, 70.858, -42.299, 143.741]
  MoveL 1962 to (54.9, -42.21, -199.64) mm, rotated rx -11.83 ry -17.7 rz 126.62 deg; joints [4.547, -32.473, 116.916, 232.183, 70.846, -42.314, 143.741]
  MoveL 1963 to (55, -42.67, -199.67) mm, rotated rx -11.83 ry -17.7 rz 126.62 deg; joints [4.539, -32.457, 116.879, 232.181, 70.832, -42.331, 143.741]
  MoveL 1964 to (55.12, -43.14, -199.69) mm, rotated rx -11.83 ry -17.7 rz 126.62 deg; joints [4.53, -32.443, 116.841, 232.179, 70.818, -42.35, 143.741]
  MoveL 1965 to (55.25, -43.63, -199.7) mm, rotated rx -11.83 ry -17.7 rz 126.62 deg; joints [4.521, -32.429, 116.803, 232.176, 70.802, -42.37, 143.741]
  MoveL 1966 to (55.39, -44.13, -199.7) mm, rotated rx -11.83 ry -17.7 rz 126.62 deg; joints [4.512, -32.415, 116.763, 232.174, 70.785, -42.391, 143.741]
  MoveL 1967 to (55.9, -47.01, -200.04) mm, rotated rx -11.83 ry -17.7 rz 126.62 deg; joints [4.467, -32.307, 116.529, 232.163, 70.704, -42.494, 143.741]
  MoveL 1968 to (55.88, -48.31, -200.47) mm, rotated rx -11.83 ry -17.7 rz 126.62 deg; joints [4.452, -32.237, 116.418, 232.159, 70.678, -42.527, 143.741]
  MoveL 1969 to (55.7, -49.52, -201.08) mm, rotated rx -11.83 ry -17.7 rz 126.62 deg; joints [4.444, -32.156, 116.312, 232.158, 70.662, -42.547, 143.741]
